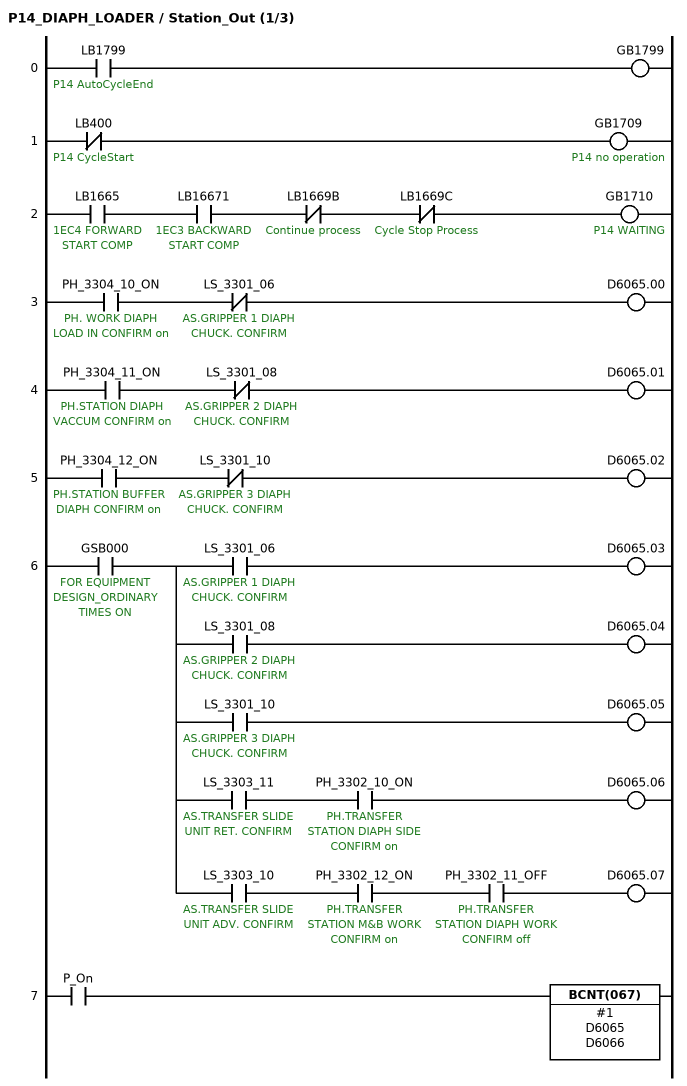
; [picture p216: P14_DIAPH_LOADER / Station_Out, rungs 0-7]
; rung 0
LD LB1799  ; P14 AutoCycleEnd
OUT GB1799
; rung 1
LDNOT LB400  ; P14 CycleStart
OUT GB1709  ; P14 no operation
; rung 2
LD LB1665  ; 1EC4 FORWARD START COMP
AND LB16671  ; 1EC3 BACKWARD START COMP
ANDNOT LB1669B  ; Continue process
ANDNOT LB1669C  ; Cycle Stop Process
OUT GB1710  ; P14 WAITING
; rung 3
LD PH_3304_10_ON  ; PH. WORK DIAPH LOAD IN CONFIRM on
ANDNOT LS_3301_06  ; AS.GRIPPER 1 DIAPH CHUCK. CONFIRM
OUT D6065.00
; rung 4
LD PH_3304_11_ON  ; PH.STATION DIAPH VACCUM CONFIRM on
ANDNOT LS_3301_08  ; AS.GRIPPER 2 DIAPH CHUCK. CONFIRM
OUT D6065.01
; rung 5
LD PH_3304_12_ON  ; PH.STATION BUFFER DIAPH CONFIRM on
ANDNOT LS_3301_10  ; AS.GRIPPER 3 DIAPH CHUCK. CONFIRM
OUT D6065.02
; rung 6
LD GSB000  ; FOR EQUIPMENT DESIGN_ORDINARY TIMES ON
OUT TR0
AND LS_3301_06  ; AS.GRIPPER 1 DIAPH CHUCK. CONFIRM
OUT D6065.03
LD TR0
AND LS_3301_08  ; AS.GRIPPER 2 DIAPH CHUCK. CONFIRM
OUT D6065.04
LD TR0
AND LS_3301_10  ; AS.GRIPPER 3 DIAPH CHUCK. CONFIRM
OUT D6065.05
LD TR0
AND LS_3303_11  ; AS.TRANSFER SLIDE UNIT RET. CONFIRM
AND PH_3302_10_ON  ; PH.TRANSFER STATION DIAPH SIDE CONFIRM on
OUT D6065.06
LD TR0
AND LS_3303_10  ; AS.TRANSFER SLIDE UNIT ADV. CONFIRM
AND PH_3302_12_ON  ; PH.TRANSFER STATION M&B WORK CONFIRM on
AND PH_3302_11_OFF  ; PH.TRANSFER STATION DIAPH WORK CONFIRM off
OUT D6065.07
; rung 7
LD P_On
BCNT(067) #1 D6065 D6066

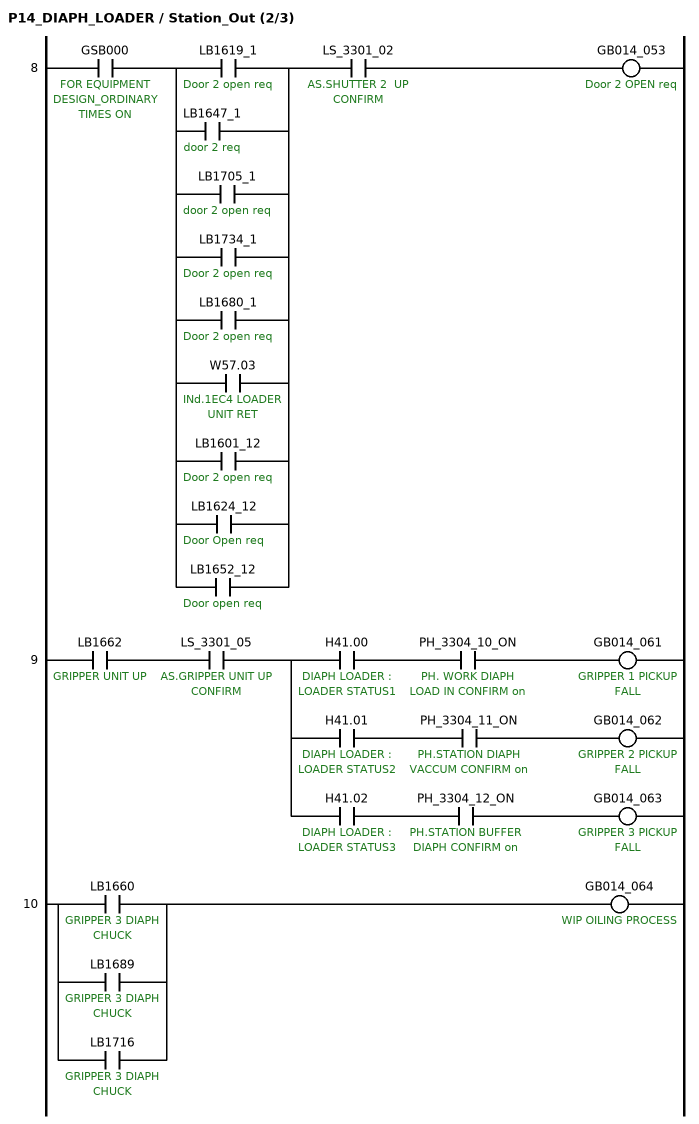
; rung 8
LD GSB000  ; FOR EQUIPMENT DESIGN_ORDINARY TIMES ON
LD LB1619_1  ; Door 2 open req
OR LB1647_1  ; door 2 req
OR LB1705_1  ; door 2 open req
OR LB1734_1  ; Door 2 open req
OR LB1680_1  ; Door 2 open req
OR W57.03  ; INd.1EC4 LOADER UNIT RET
OR LB1601_12  ; Door 2 open req
OR LB1624_12  ; Door Open req
OR LB1652_12  ; Door open req
ANDLD
AND LS_3301_02  ; AS.SHUTTER 2  UP CONFIRM
OUT GB014_053  ; Door 2 OPEN req
; rung 9
LD LB1662  ; GRIPPER UNIT UP
AND LS_3301_05  ; AS.GRIPPER UNIT UP CONFIRM
OUT TR0
AND H41.00  ; DIAPH LOADER : LOADER STATUS1
AND PH_3304_10_ON  ; PH. WORK DIAPH LOAD IN CONFIRM on
OUT GB014_061  ; GRIPPER 1 PICKUP FALL
LD TR0
AND H41.01  ; DIAPH LOADER : LOADER STATUS2
AND PH_3304_11_ON  ; PH.STATION DIAPH VACCUM CONFIRM on
OUT GB014_062  ; GRIPPER 2 PICKUP FALL
LD TR0
AND H41.02  ; DIAPH LOADER : LOADER STATUS3
AND PH_3304_12_ON  ; PH.STATION BUFFER DIAPH CONFIRM on
OUT GB014_063  ; GRIPPER 3 PICKUP FALL
; rung 10
LD LB1660  ; GRIPPER 3 DIAPH CHUCK
OR LB1689  ; GRIPPER 3 DIAPH CHUCK
OR LB1716  ; GRIPPER 3 DIAPH CHUCK
OUT GB014_064  ; WIP OILING PROCESS

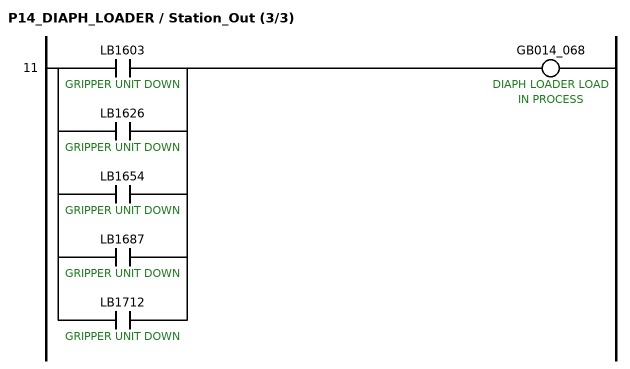
; rung 11
LD LB1603  ; GRIPPER UNIT DOWN
OR LB1626  ; GRIPPER UNIT DOWN
OR LB1654  ; GRIPPER UNIT DOWN
OR LB1687  ; GRIPPER UNIT DOWN
OR LB1712  ; GRIPPER UNIT DOWN
OUT GB014_068  ; DIAPH LOADER LOAD IN PROCESS

### Section Individual

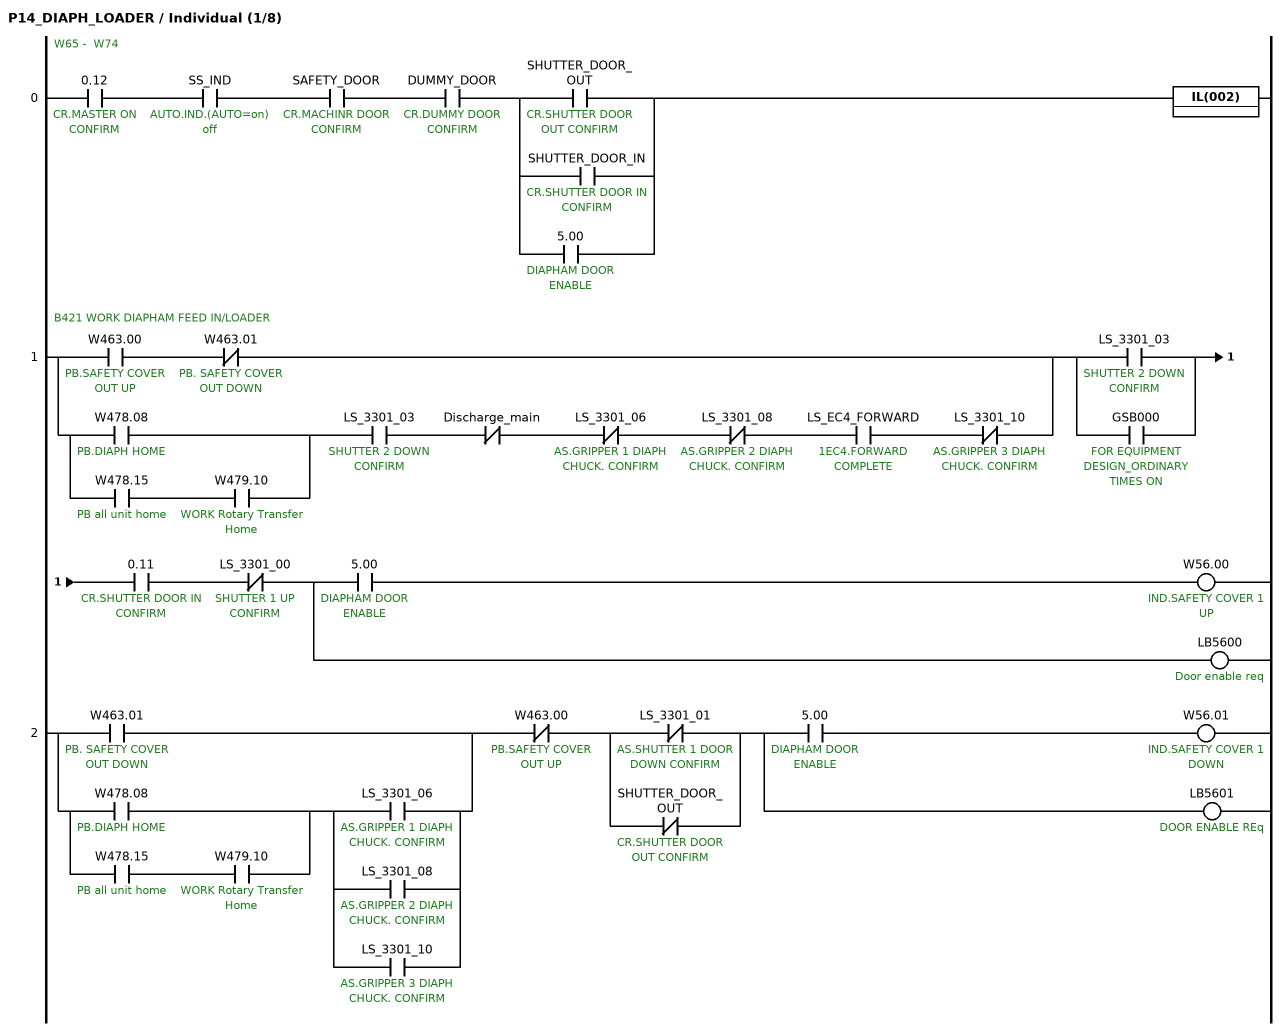
; rung 0: W65 -  W74
LD 0.12  ; CR.MASTER ON CONFIRM
AND SS_IND  ; AUTO.IND.(AUTO=on) off
AND SAFETY_DOOR  ; CR.MACHINR DOOR CONFIRM
AND DUMMY_DOOR  ; CR.DUMMY DOOR CONFIRM
LD SHUTTER_DOOR_OUT  ; CR.SHUTTER DOOR OUT CONFIRM
OR SHUTTER_DOOR_IN  ; CR.SHUTTER DOOR IN CONFIRM
OR 5.00  ; DIAPHAM DOOR ENABLE
ANDLD
IL(002)
; rung 1: B421 WORK DIAPHAM FEED IN/LOADER
LD W463.00  ; PB.SAFETY COVER OUT UP
ANDNOT W463.01  ; PB. SAFETY COVER OUT DOWN
LD W478.08  ; PB.DIAPH HOME
LD W478.15  ; PB all unit home
AND W479.10  ; WORK Rotary Transfer Home
ORLD
AND LS_3301_03  ; SHUTTER 2 DOWN CONFIRM
ANDNOT Discharge_main
ANDNOT LS_3301_06  ; AS.GRIPPER 1 DIAPH CHUCK. CONFIRM
ANDNOT LS_3301_08  ; AS.GRIPPER 2 DIAPH CHUCK. CONFIRM
AND LS_EC4_FORWARD  ; 1EC4.FORWARD COMPLETE
ANDNOT LS_3301_10  ; AS.GRIPPER 3 DIAPH CHUCK. CONFIRM
ORLD
LD LS_3301_03  ; SHUTTER 2 DOWN CONFIRM
OR GSB000  ; FOR EQUIPMENT DESIGN_ORDINARY TIMES ON
ANDLD
AND 0.11  ; CR.SHUTTER DOOR IN CONFIRM
ANDNOT LS_3301_00  ; SHUTTER 1 UP CONFIRM
OUT TR0
AND 5.00  ; DIAPHAM DOOR ENABLE
OUT W56.00  ; IND.SAFETY COVER 1 UP
LD TR0
OUT LB5600  ; Door enable req
; rung 2
LD W463.01  ; PB. SAFETY COVER OUT DOWN
LD W478.08  ; PB.DIAPH HOME
LD W478.15  ; PB all unit home
AND W479.10  ; WORK Rotary Transfer Home
ORLD
LD LS_3301_06  ; AS.GRIPPER 1 DIAPH CHUCK. CONFIRM
OR LS_3301_08  ; AS.GRIPPER 2 DIAPH CHUCK. CONFIRM
OR LS_3301_10  ; AS.GRIPPER 3 DIAPH CHUCK. CONFIRM
ANDLD
ORLD
ANDNOT W463.00  ; PB.SAFETY COVER OUT UP
LDNOT LS_3301_01  ; AS.SHUTTER 1 DOOR DOWN CONFIRM
ORNOT SHUTTER_DOOR_OUT  ; CR.SHUTTER DOOR OUT CONFIRM
ANDLD
OUT TR0
AND 5.00  ; DIAPHAM DOOR ENABLE
OUT W56.01  ; IND.SAFETY COVER 1 DOWN
LD TR0
OUT LB5601  ; DOOR ENABLE REq

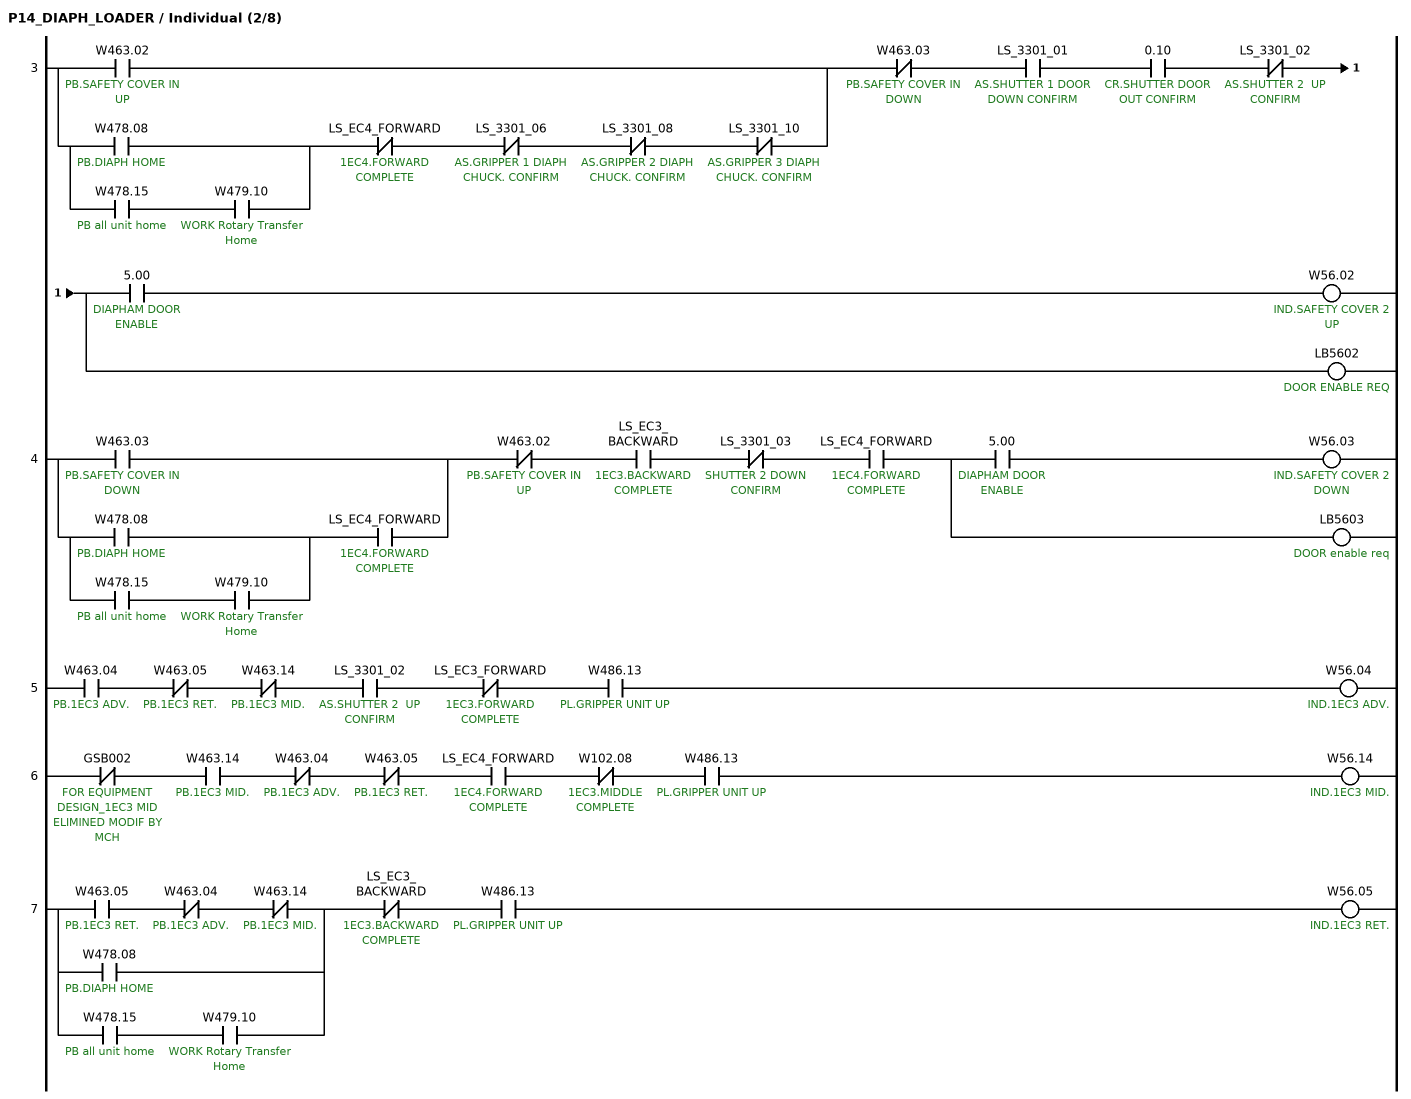
; rung 3
LD W463.02  ; PB.SAFETY COVER IN UP
LD W478.08  ; PB.DIAPH HOME
LD W478.15  ; PB all unit home
AND W479.10  ; WORK Rotary Transfer Home
ORLD
ANDNOT LS_EC4_FORWARD  ; 1EC4.FORWARD COMPLETE
ANDNOT LS_3301_06  ; AS.GRIPPER 1 DIAPH CHUCK. CONFIRM
ANDNOT LS_3301_08  ; AS.GRIPPER 2 DIAPH CHUCK. CONFIRM
ANDNOT LS_3301_10  ; AS.GRIPPER 3 DIAPH CHUCK. CONFIRM
ORLD
ANDNOT W463.03  ; PB.SAFETY COVER IN DOWN
AND LS_3301_01  ; AS.SHUTTER 1 DOOR DOWN CONFIRM
AND 0.10  ; CR.SHUTTER DOOR OUT CONFIRM
ANDNOT LS_3301_02  ; AS.SHUTTER 2  UP CONFIRM
OUT TR0
AND 5.00  ; DIAPHAM DOOR ENABLE
OUT W56.02  ; IND.SAFETY COVER 2 UP
LD TR0
OUT LB5602  ; DOOR ENABLE REQ
; rung 4
LD W463.03  ; PB.SAFETY COVER IN DOWN
LD W478.08  ; PB.DIAPH HOME
LD W478.15  ; PB all unit home
AND W479.10  ; WORK Rotary Transfer Home
ORLD
AND LS_EC4_FORWARD  ; 1EC4.FORWARD COMPLETE
ORLD
ANDNOT W463.02  ; PB.SAFETY COVER IN UP
AND LS_EC3_BACKWARD  ; 1EC3.BACKWARD COMPLETE
ANDNOT LS_3301_03  ; SHUTTER 2 DOWN CONFIRM
AND LS_EC4_FORWARD  ; 1EC4.FORWARD COMPLETE
OUT TR0
AND 5.00  ; DIAPHAM DOOR ENABLE
OUT W56.03  ; IND.SAFETY COVER 2 DOWN
LD TR0
OUT LB5603  ; DOOR enable req
; rung 5
LD W463.04  ; PB.1EC3 ADV.
ANDNOT W463.05  ; PB.1EC3 RET.
ANDNOT W463.14  ; PB.1EC3 MID.
AND LS_3301_02  ; AS.SHUTTER 2  UP CONFIRM
ANDNOT LS_EC3_FORWARD  ; 1EC3.FORWARD COMPLETE
AND W486.13  ; PL.GRIPPER UNIT UP
OUT W56.04  ; IND.1EC3 ADV.
; rung 6
LDNOT GSB002  ; FOR EQUIPMENT DESIGN_1EC3 MID ELIMINED MODIF BY MCH
AND W463.14  ; PB.1EC3 MID.
ANDNOT W463.04  ; PB.1EC3 ADV.
ANDNOT W463.05  ; PB.1EC3 RET.
AND LS_EC4_FORWARD  ; 1EC4.FORWARD COMPLETE
ANDNOT W102.08  ; 1EC3.MIDDLE COMPLETE
AND W486.13  ; PL.GRIPPER UNIT UP
OUT W56.14  ; IND.1EC3 MID.
; rung 7
LD W463.05  ; PB.1EC3 RET.
ANDNOT W463.04  ; PB.1EC3 ADV.
ANDNOT W463.14  ; PB.1EC3 MID.
LD W478.08  ; PB.DIAPH HOME
LD W478.15  ; PB all unit home
AND W479.10  ; WORK Rotary Transfer Home
ORLD
ORLD
ANDNOT LS_EC3_BACKWARD  ; 1EC3.BACKWARD COMPLETE
AND W486.13  ; PL.GRIPPER UNIT UP
OUT W56.05  ; IND.1EC3 RET.

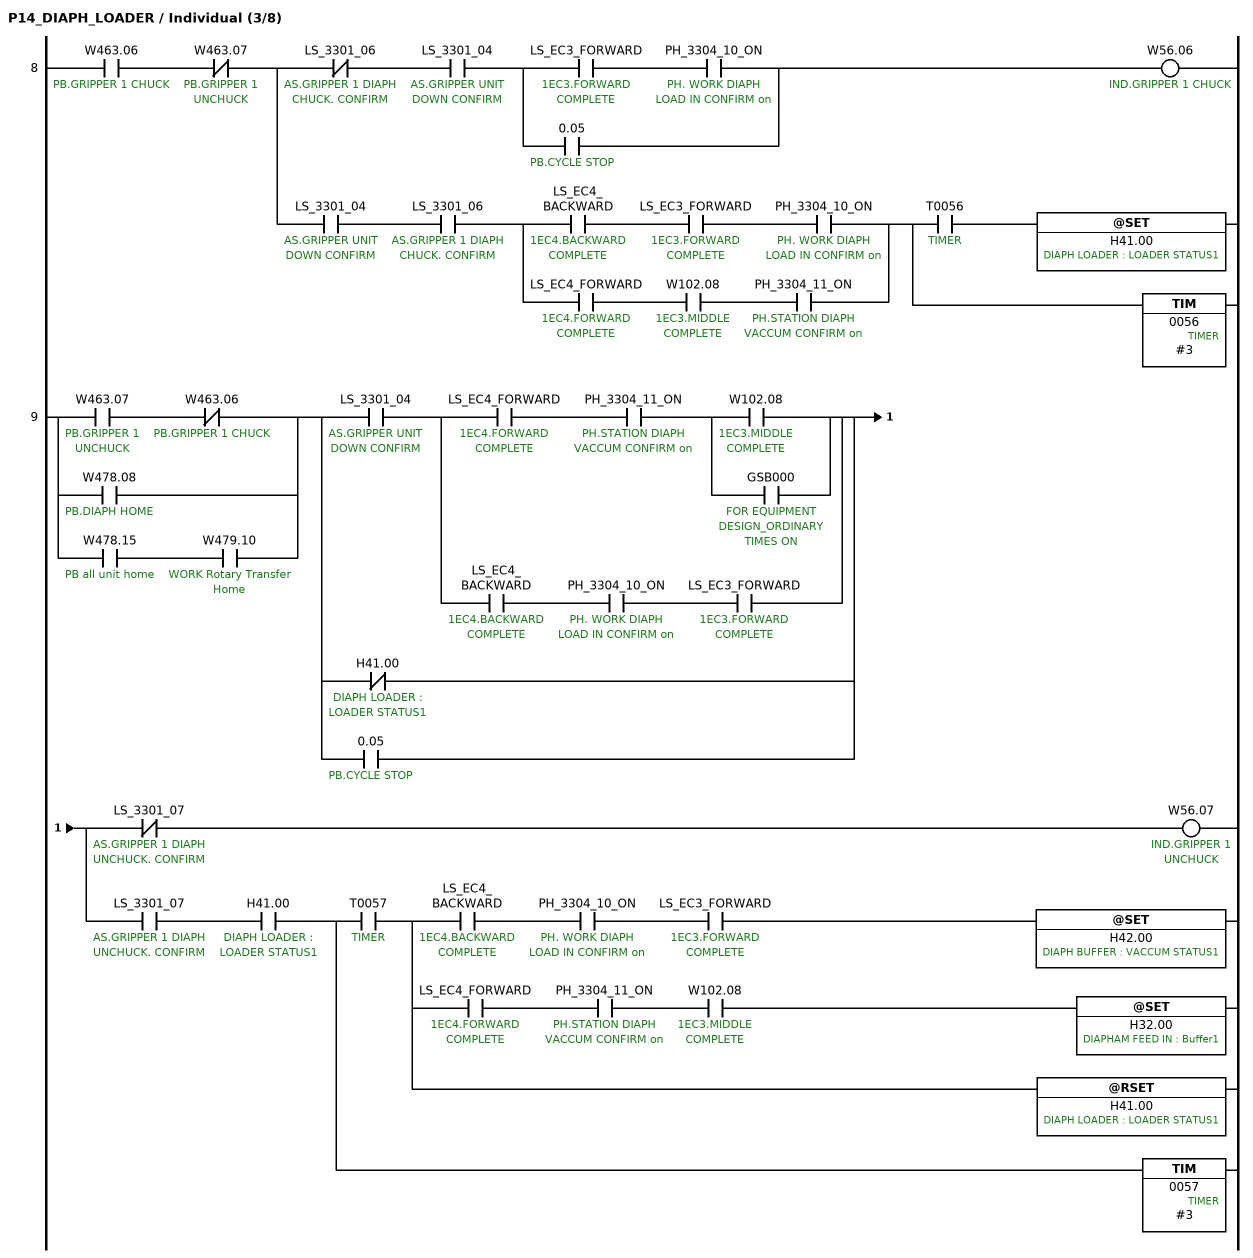
; rung 8
LD W463.06  ; PB.GRIPPER 1 CHUCK
ANDNOT W463.07  ; PB.GRIPPER 1 UNCHUCK
OUT TR0
ANDNOT LS_3301_06  ; AS.GRIPPER 1 DIAPH CHUCK. CONFIRM
AND LS_3301_04  ; AS.GRIPPER UNIT DOWN CONFIRM
LD LS_EC3_FORWARD  ; 1EC3.FORWARD COMPLETE
AND PH_3304_10_ON  ; PH. WORK DIAPH LOAD IN CONFIRM on
OR 0.05  ; PB.CYCLE STOP
ANDLD
OUT W56.06  ; IND.GRIPPER 1 CHUCK
LD TR0
AND LS_3301_04  ; AS.GRIPPER UNIT DOWN CONFIRM
AND LS_3301_06  ; AS.GRIPPER 1 DIAPH CHUCK. CONFIRM
LD LS_EC4_BACKWARD  ; 1EC4.BACKWARD COMPLETE
AND LS_EC3_FORWARD  ; 1EC3.FORWARD COMPLETE
AND PH_3304_10_ON  ; PH. WORK DIAPH LOAD IN CONFIRM on
LD LS_EC4_FORWARD  ; 1EC4.FORWARD COMPLETE
AND W102.08  ; 1EC3.MIDDLE COMPLETE
AND PH_3304_11_ON  ; PH.STATION DIAPH VACCUM CONFIRM on
ORLD
ANDLD
OUT TR0
AND T0056  ; TIMER
@SET H41.00  ; DIAPH LOADER : LOADER STATUS1
LD TR0
TIM 0056 #3  ; TIMER
; rung 9
LD W463.07  ; PB.GRIPPER 1 UNCHUCK
ANDNOT W463.06  ; PB.GRIPPER 1 CHUCK
OR W478.08  ; PB.DIAPH HOME
LD W478.15  ; PB all unit home
AND W479.10  ; WORK Rotary Transfer Home
ORLD
LD LS_3301_04  ; AS.GRIPPER UNIT DOWN CONFIRM
LD LS_EC4_FORWARD  ; 1EC4.FORWARD COMPLETE
AND PH_3304_11_ON  ; PH.STATION DIAPH VACCUM CONFIRM on
LD W102.08  ; 1EC3.MIDDLE COMPLETE
OR GSB000  ; FOR EQUIPMENT DESIGN_ORDINARY TIMES ON
ANDLD
LD LS_EC4_BACKWARD  ; 1EC4.BACKWARD COMPLETE
AND PH_3304_10_ON  ; PH. WORK DIAPH LOAD IN CONFIRM on
AND LS_EC3_FORWARD  ; 1EC3.FORWARD COMPLETE
ORLD
ANDLD
ORNOT H41.00  ; DIAPH LOADER : LOADER STATUS1
OR 0.05  ; PB.CYCLE STOP
ANDLD
OUT TR0
ANDNOT LS_3301_07  ; AS.GRIPPER 1 DIAPH UNCHUCK. CONFIRM
OUT W56.07  ; IND.GRIPPER 1 UNCHUCK
LD TR0
AND LS_3301_07  ; AS.GRIPPER 1 DIAPH UNCHUCK. CONFIRM
AND H41.00  ; DIAPH LOADER : LOADER STATUS1
OUT TR0
AND T0057  ; TIMER
OUT TR1
AND LS_EC4_BACKWARD  ; 1EC4.BACKWARD COMPLETE
AND PH_3304_10_ON  ; PH. WORK DIAPH LOAD IN CONFIRM on
AND LS_EC3_FORWARD  ; 1EC3.FORWARD COMPLETE
@SET H42.00  ; DIAPH BUFFER : VACCUM STATUS1
LD TR1
AND LS_EC4_FORWARD  ; 1EC4.FORWARD COMPLETE
AND PH_3304_11_ON  ; PH.STATION DIAPH VACCUM CONFIRM on
AND W102.08  ; 1EC3.MIDDLE COMPLETE
@SET H32.00  ; DIAPHAM FEED IN : Buffer1
LD TR1
@RSET H41.00  ; DIAPH LOADER : LOADER STATUS1
LD TR0
TIM 0057 #3  ; TIMER

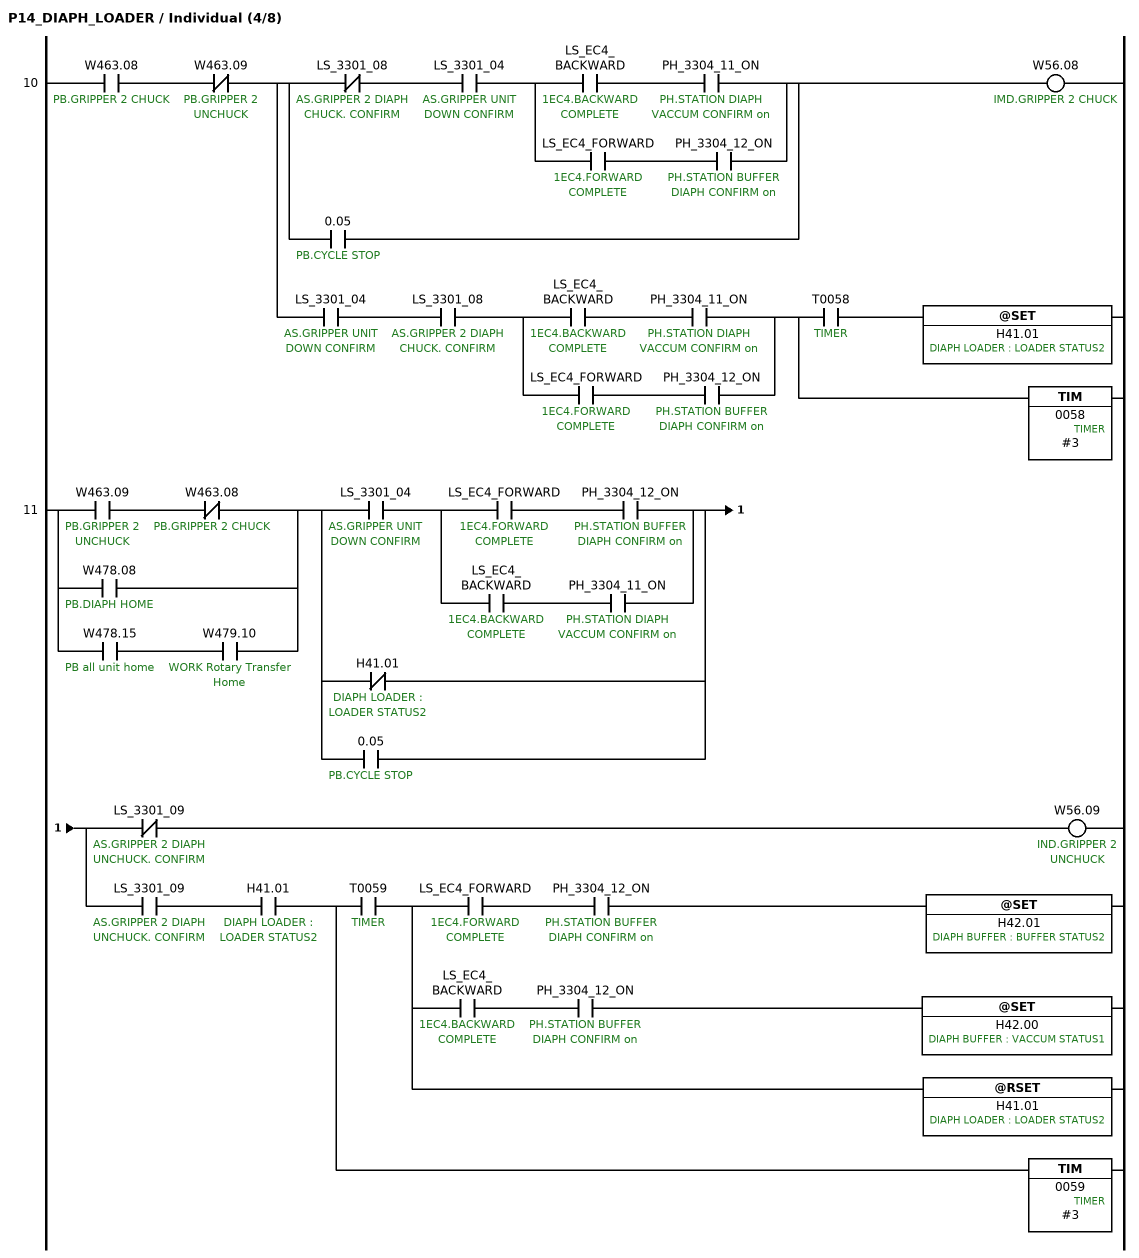
; rung 10
LD W463.08  ; PB.GRIPPER 2 CHUCK
ANDNOT W463.09  ; PB.GRIPPER 2 UNCHUCK
OUT TR0
LDNOT LS_3301_08  ; AS.GRIPPER 2 DIAPH CHUCK. CONFIRM
AND LS_3301_04  ; AS.GRIPPER UNIT DOWN CONFIRM
LD LS_EC4_BACKWARD  ; 1EC4.BACKWARD COMPLETE
AND PH_3304_11_ON  ; PH.STATION DIAPH VACCUM CONFIRM on
LD LS_EC4_FORWARD  ; 1EC4.FORWARD COMPLETE
AND PH_3304_12_ON  ; PH.STATION BUFFER DIAPH CONFIRM on
ORLD
ANDLD
OR 0.05  ; PB.CYCLE STOP
ANDLD
OUT W56.08  ; IMD.GRIPPER 2 CHUCK
LD TR0
AND LS_3301_04  ; AS.GRIPPER UNIT DOWN CONFIRM
AND LS_3301_08  ; AS.GRIPPER 2 DIAPH CHUCK. CONFIRM
LD LS_EC4_BACKWARD  ; 1EC4.BACKWARD COMPLETE
AND PH_3304_11_ON  ; PH.STATION DIAPH VACCUM CONFIRM on
LD LS_EC4_FORWARD  ; 1EC4.FORWARD COMPLETE
AND PH_3304_12_ON  ; PH.STATION BUFFER DIAPH CONFIRM on
ORLD
ANDLD
OUT TR0
AND T0058  ; TIMER
@SET H41.01  ; DIAPH LOADER : LOADER STATUS2
LD TR0
TIM 0058 #3  ; TIMER
; rung 11
LD W463.09  ; PB.GRIPPER 2 UNCHUCK
ANDNOT W463.08  ; PB.GRIPPER 2 CHUCK
OR W478.08  ; PB.DIAPH HOME
LD W478.15  ; PB all unit home
AND W479.10  ; WORK Rotary Transfer Home
ORLD
LD LS_3301_04  ; AS.GRIPPER UNIT DOWN CONFIRM
LD LS_EC4_FORWARD  ; 1EC4.FORWARD COMPLETE
AND PH_3304_12_ON  ; PH.STATION BUFFER DIAPH CONFIRM on
LD LS_EC4_BACKWARD  ; 1EC4.BACKWARD COMPLETE
AND PH_3304_11_ON  ; PH.STATION DIAPH VACCUM CONFIRM on
ORLD
ANDLD
ORNOT H41.01  ; DIAPH LOADER : LOADER STATUS2
OR 0.05  ; PB.CYCLE STOP
ANDLD
OUT TR0
ANDNOT LS_3301_09  ; AS.GRIPPER 2 DIAPH UNCHUCK. CONFIRM
OUT W56.09  ; IND.GRIPPER 2 UNCHUCK
LD TR0
AND LS_3301_09  ; AS.GRIPPER 2 DIAPH UNCHUCK. CONFIRM
AND H41.01  ; DIAPH LOADER : LOADER STATUS2
OUT TR0
AND T0059  ; TIMER
OUT TR1
AND LS_EC4_FORWARD  ; 1EC4.FORWARD COMPLETE
AND PH_3304_12_ON  ; PH.STATION BUFFER DIAPH CONFIRM on
@SET H42.01  ; DIAPH BUFFER : BUFFER STATUS2
LD TR1
AND LS_EC4_BACKWARD  ; 1EC4.BACKWARD COMPLETE
AND PH_3304_12_ON  ; PH.STATION BUFFER DIAPH CONFIRM on
@SET H42.00  ; DIAPH BUFFER : VACCUM STATUS1
LD TR1
@RSET H41.01  ; DIAPH LOADER : LOADER STATUS2
LD TR0
TIM 0059 #3  ; TIMER

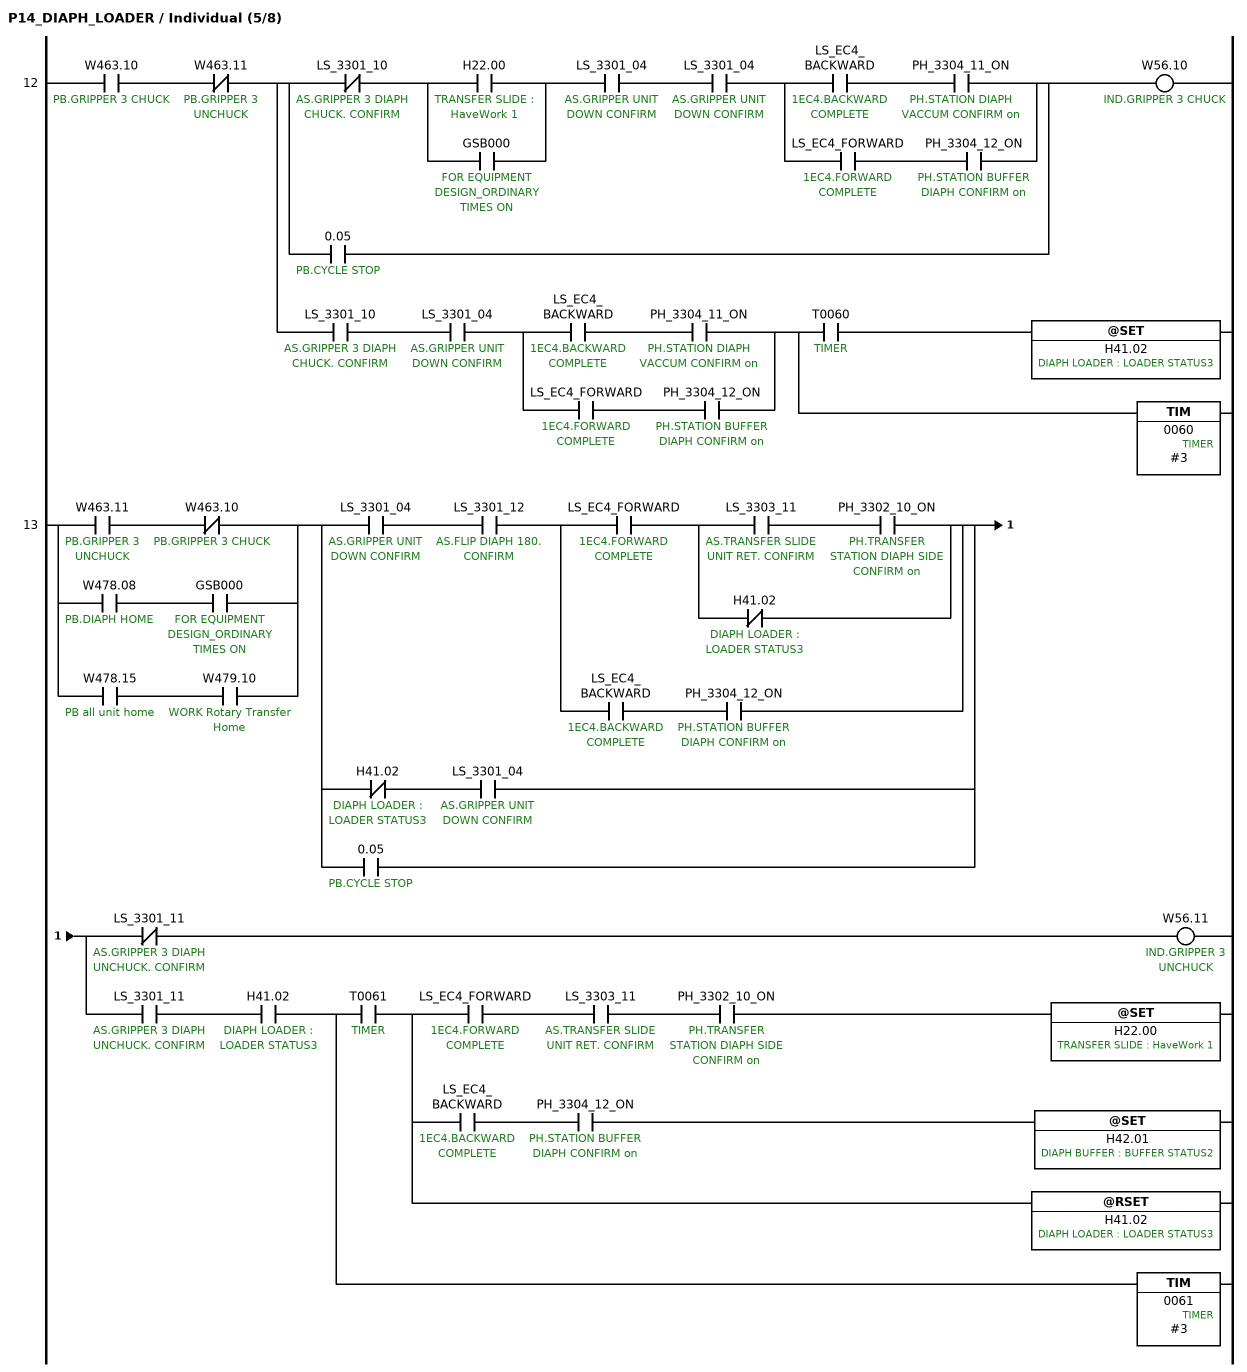
; rung 12
LD W463.10  ; PB.GRIPPER 3 CHUCK
ANDNOT W463.11  ; PB.GRIPPER 3 UNCHUCK
OUT TR0
LDNOT LS_3301_10  ; AS.GRIPPER 3 DIAPH CHUCK. CONFIRM
LD H22.00  ; TRANSFER SLIDE : HaveWork 1
OR GSB000  ; FOR EQUIPMENT DESIGN_ORDINARY TIMES ON
ANDLD
AND LS_3301_04  ; AS.GRIPPER UNIT DOWN CONFIRM  // PROHIBIT LOAD WORK FORM TRANSFER UNIT
AND LS_3301_04  ; AS.GRIPPER UNIT DOWN CONFIRM
LD LS_EC4_BACKWARD  ; 1EC4.BACKWARD COMPLETE
AND PH_3304_11_ON  ; PH.STATION DIAPH VACCUM CONFIRM on
LD LS_EC4_FORWARD  ; 1EC4.FORWARD COMPLETE
AND PH_3304_12_ON  ; PH.STATION BUFFER DIAPH CONFIRM on
ORLD
ANDLD
OR 0.05  ; PB.CYCLE STOP
ANDLD
OUT W56.10  ; IND.GRIPPER 3 CHUCK
LD TR0
AND LS_3301_10  ; AS.GRIPPER 3 DIAPH CHUCK. CONFIRM
AND LS_3301_04  ; AS.GRIPPER UNIT DOWN CONFIRM
LD LS_EC4_BACKWARD  ; 1EC4.BACKWARD COMPLETE
AND PH_3304_11_ON  ; PH.STATION DIAPH VACCUM CONFIRM on
LD LS_EC4_FORWARD  ; 1EC4.FORWARD COMPLETE
AND PH_3304_12_ON  ; PH.STATION BUFFER DIAPH CONFIRM on
ORLD
ANDLD
OUT TR0
AND T0060  ; TIMER
@SET H41.02  ; DIAPH LOADER : LOADER STATUS3
LD TR0
TIM 0060 #3  ; TIMER
; rung 13
LD W463.11  ; PB.GRIPPER 3 UNCHUCK
ANDNOT W463.10  ; PB.GRIPPER 3 CHUCK
LD W478.08  ; PB.DIAPH HOME
AND GSB000  ; FOR EQUIPMENT DESIGN_ORDINARY TIMES ON
ORLD
LD W478.15  ; PB all unit home
AND W479.10  ; WORK Rotary Transfer Home
ORLD
LD LS_3301_04  ; AS.GRIPPER UNIT DOWN CONFIRM
AND LS_3301_12  ; AS.FLIP DIAPH 180. CONFIRM
LD LS_EC4_FORWARD  ; 1EC4.FORWARD COMPLETE
LD LS_3303_11  ; AS.TRANSFER SLIDE UNIT RET. CONFIRM
AND PH_3302_10_ON  ; PH.TRANSFER STATION DIAPH SIDE CONFIRM on
ORNOT H41.02  ; DIAPH LOADER : LOADER STATUS3
ANDLD
LD LS_EC4_BACKWARD  ; 1EC4.BACKWARD COMPLETE
AND PH_3304_12_ON  ; PH.STATION BUFFER DIAPH CONFIRM on
ORLD
ANDLD
LDNOT H41.02  ; DIAPH LOADER : LOADER STATUS3
AND LS_3301_04  ; AS.GRIPPER UNIT DOWN CONFIRM
ORLD
OR 0.05  ; PB.CYCLE STOP
ANDLD
OUT TR0
ANDNOT LS_3301_11  ; AS.GRIPPER 3 DIAPH UNCHUCK. CONFIRM
OUT W56.11  ; IND.GRIPPER 3 UNCHUCK
LD TR0
AND LS_3301_11  ; AS.GRIPPER 3 DIAPH UNCHUCK. CONFIRM
AND H41.02  ; DIAPH LOADER : LOADER STATUS3
OUT TR0
AND T0061  ; TIMER
OUT TR1
AND LS_EC4_FORWARD  ; 1EC4.FORWARD COMPLETE
AND LS_3303_11  ; AS.TRANSFER SLIDE UNIT RET. CONFIRM
AND PH_3302_10_ON  ; PH.TRANSFER STATION DIAPH SIDE CONFIRM on
@SET H22.00  ; TRANSFER SLIDE : HaveWork 1
LD TR1
AND LS_EC4_BACKWARD  ; 1EC4.BACKWARD COMPLETE
AND PH_3304_12_ON  ; PH.STATION BUFFER DIAPH CONFIRM on
@SET H42.01  ; DIAPH BUFFER : BUFFER STATUS2
LD TR1
@RSET H41.02  ; DIAPH LOADER : LOADER STATUS3
LD TR0
TIM 0061 #3  ; TIMER

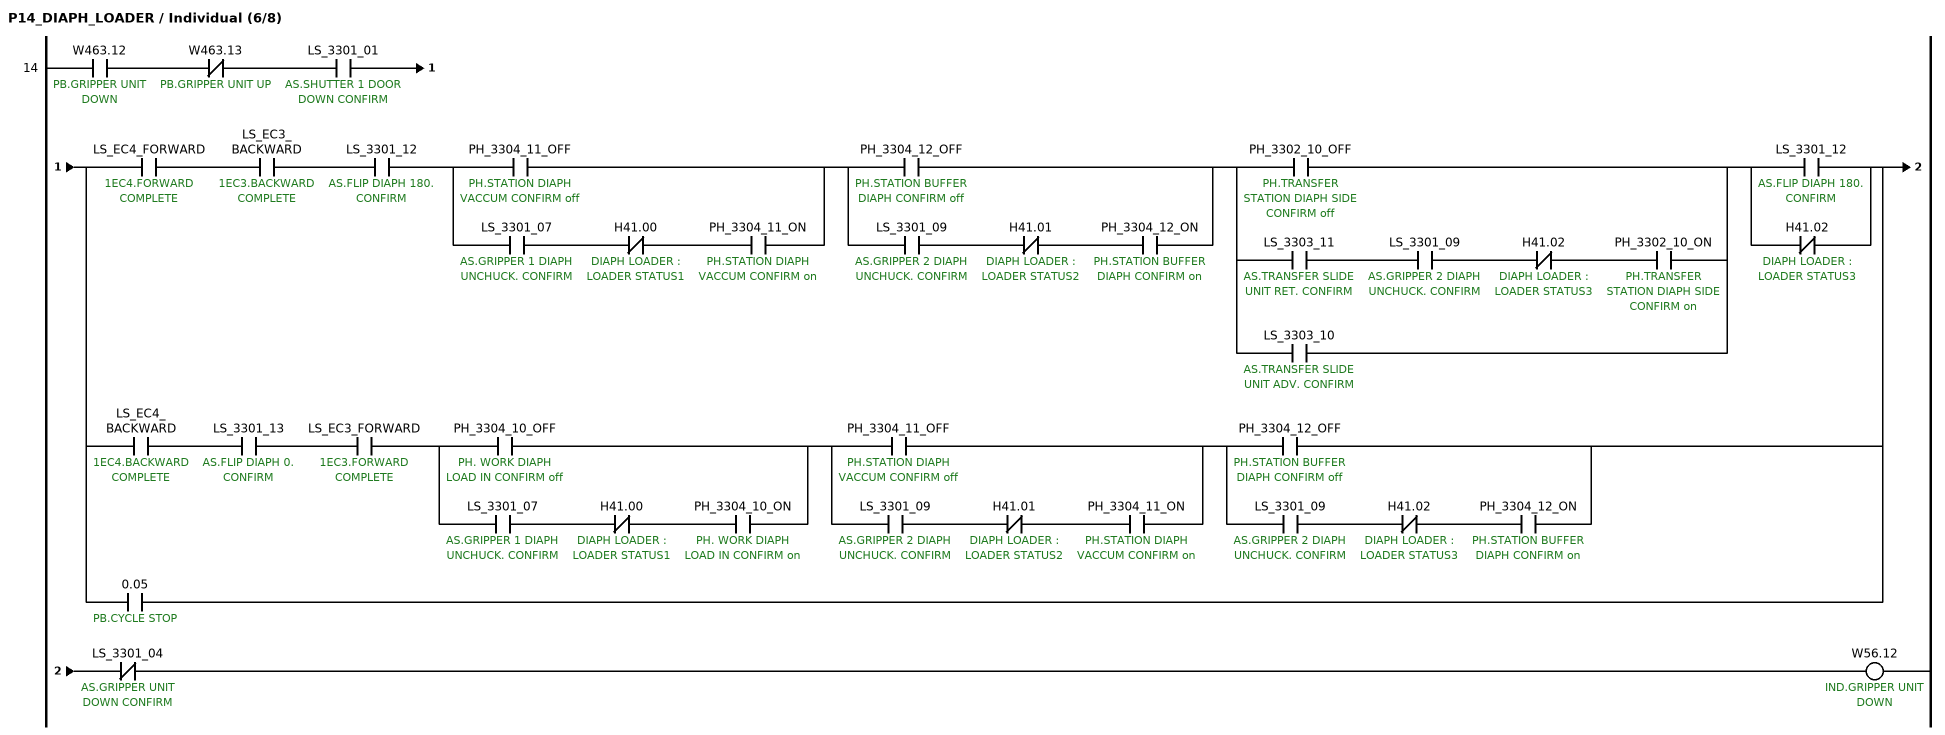
; rung 14
LD W463.12  ; PB.GRIPPER UNIT DOWN
ANDNOT W463.13  ; PB.GRIPPER UNIT UP
AND LS_3301_01  ; AS.SHUTTER 1 DOOR DOWN CONFIRM
LD LS_EC4_FORWARD  ; 1EC4.FORWARD COMPLETE
AND LS_EC3_BACKWARD  ; 1EC3.BACKWARD COMPLETE
AND LS_3301_12  ; AS.FLIP DIAPH 180. CONFIRM
LD PH_3304_11_OFF  ; PH.STATION DIAPH VACCUM CONFIRM off
LD LS_3301_07  ; AS.GRIPPER 1 DIAPH UNCHUCK. CONFIRM
ANDNOT H41.00  ; DIAPH LOADER : LOADER STATUS1
AND PH_3304_11_ON  ; PH.STATION DIAPH VACCUM CONFIRM on
ORLD
ANDLD
LD PH_3304_12_OFF  ; PH.STATION BUFFER DIAPH CONFIRM off
LD LS_3301_09  ; AS.GRIPPER 2 DIAPH UNCHUCK. CONFIRM
ANDNOT H41.01  ; DIAPH LOADER : LOADER STATUS2
AND PH_3304_12_ON  ; PH.STATION BUFFER DIAPH CONFIRM on
ORLD
ANDLD
LD PH_3302_10_OFF  ; PH.TRANSFER STATION DIAPH SIDE CONFIRM off
LD LS_3303_11  ; AS.TRANSFER SLIDE UNIT RET. CONFIRM
AND LS_3301_09  ; AS.GRIPPER 2 DIAPH UNCHUCK. CONFIRM
ANDNOT H41.02  ; DIAPH LOADER : LOADER STATUS3
AND PH_3302_10_ON  ; PH.TRANSFER STATION DIAPH SIDE CONFIRM on
ORLD
OR LS_3303_10  ; AS.TRANSFER SLIDE UNIT ADV. CONFIRM
ANDLD
LD LS_3301_12  ; AS.FLIP DIAPH 180. CONFIRM
ORNOT H41.02  ; DIAPH LOADER : LOADER STATUS3
ANDLD
LD LS_EC4_BACKWARD  ; 1EC4.BACKWARD COMPLETE
AND LS_3301_13  ; AS.FLIP DIAPH 0. CONFIRM
AND LS_EC3_FORWARD  ; 1EC3.FORWARD COMPLETE
LD PH_3304_10_OFF  ; PH. WORK DIAPH LOAD IN CONFIRM off
LD LS_3301_07  ; AS.GRIPPER 1 DIAPH UNCHUCK. CONFIRM
ANDNOT H41.00  ; DIAPH LOADER : LOADER STATUS1
AND PH_3304_10_ON  ; PH. WORK DIAPH LOAD IN CONFIRM on
ORLD
ANDLD
LD PH_3304_11_OFF  ; PH.STATION DIAPH VACCUM CONFIRM off
LD LS_3301_09  ; AS.GRIPPER 2 DIAPH UNCHUCK. CONFIRM
ANDNOT H41.01  ; DIAPH LOADER : LOADER STATUS2
AND PH_3304_11_ON  ; PH.STATION DIAPH VACCUM CONFIRM on
ORLD
ANDLD
LD PH_3304_12_OFF  ; PH.STATION BUFFER DIAPH CONFIRM off
LD LS_3301_09  ; AS.GRIPPER 2 DIAPH UNCHUCK. CONFIRM
ANDNOT H41.02  ; DIAPH LOADER : LOADER STATUS3
AND PH_3304_12_ON  ; PH.STATION BUFFER DIAPH CONFIRM on
ORLD
ANDLD
ORLD
OR 0.05  ; PB.CYCLE STOP
ANDLD
ANDNOT LS_3301_04  ; AS.GRIPPER UNIT DOWN CONFIRM
OUT W56.12  ; IND.GRIPPER UNIT DOWN

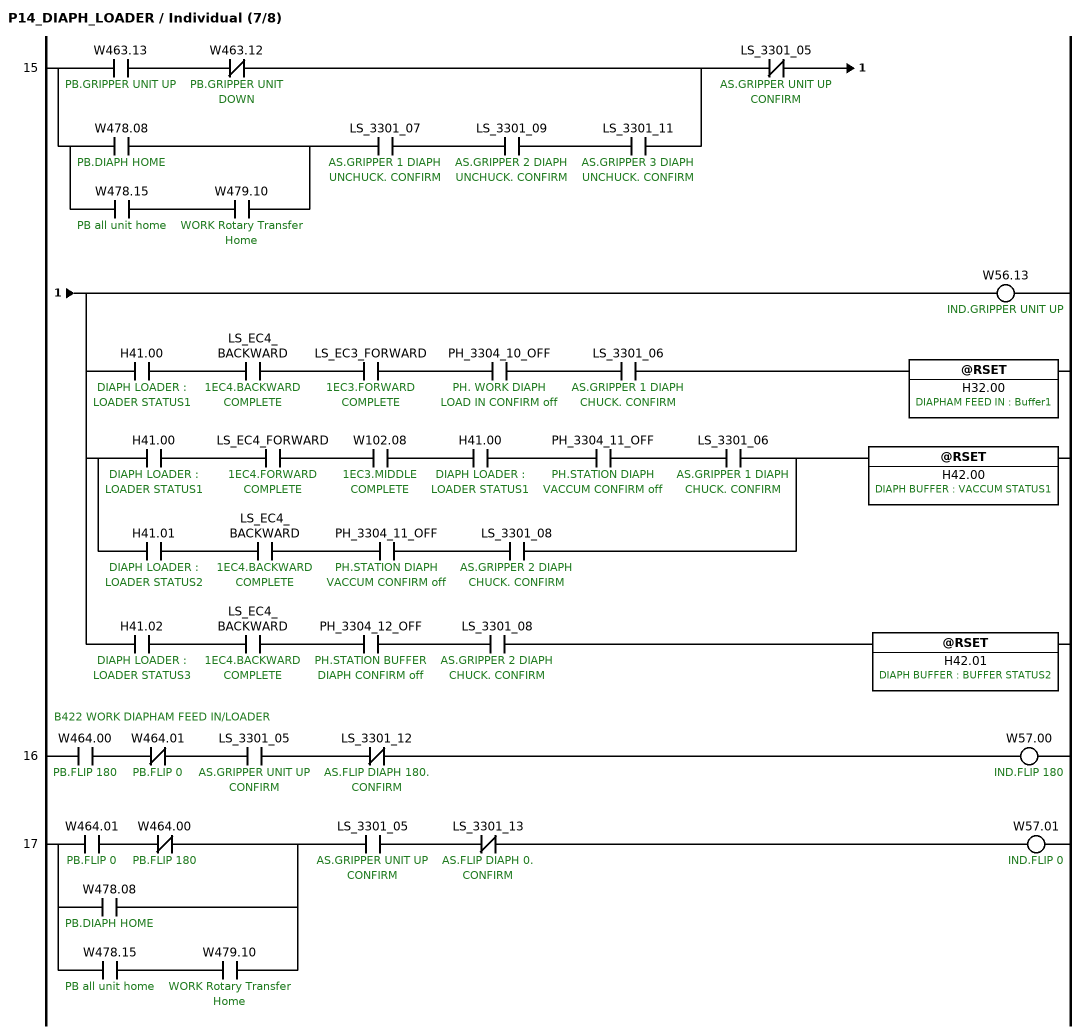
; rung 15
LD W463.13  ; PB.GRIPPER UNIT UP
ANDNOT W463.12  ; PB.GRIPPER UNIT DOWN
LD W478.08  ; PB.DIAPH HOME
LD W478.15  ; PB all unit home
AND W479.10  ; WORK Rotary Transfer Home
ORLD
AND LS_3301_07  ; AS.GRIPPER 1 DIAPH UNCHUCK. CONFIRM
AND LS_3301_09  ; AS.GRIPPER 2 DIAPH UNCHUCK. CONFIRM
AND LS_3301_11  ; AS.GRIPPER 3 DIAPH UNCHUCK. CONFIRM
ORLD
ANDNOT LS_3301_05  ; AS.GRIPPER UNIT UP CONFIRM
OUT TR0
OUT W56.13  ; IND.GRIPPER UNIT UP
AND H41.00  ; DIAPH LOADER : LOADER STATUS1
AND LS_EC4_BACKWARD  ; 1EC4.BACKWARD COMPLETE
AND LS_EC3_FORWARD  ; 1EC3.FORWARD COMPLETE
AND PH_3304_10_OFF  ; PH. WORK DIAPH LOAD IN CONFIRM off
AND LS_3301_06  ; AS.GRIPPER 1 DIAPH CHUCK. CONFIRM
@RSET H32.00  ; DIAPHAM FEED IN : Buffer1
LD TR0
LD H41.00  ; DIAPH LOADER : LOADER STATUS1
AND LS_EC4_FORWARD  ; 1EC4.FORWARD COMPLETE
AND W102.08  ; 1EC3.MIDDLE COMPLETE
AND H41.00  ; DIAPH LOADER : LOADER STATUS1
AND PH_3304_11_OFF  ; PH.STATION DIAPH VACCUM CONFIRM off
AND LS_3301_06  ; AS.GRIPPER 1 DIAPH CHUCK. CONFIRM
LD H41.01  ; DIAPH LOADER : LOADER STATUS2
AND LS_EC4_BACKWARD  ; 1EC4.BACKWARD COMPLETE
AND PH_3304_11_OFF  ; PH.STATION DIAPH VACCUM CONFIRM off
AND LS_3301_08  ; AS.GRIPPER 2 DIAPH CHUCK. CONFIRM
ORLD
ANDLD
@RSET H42.00  ; DIAPH BUFFER : VACCUM STATUS1
LD TR0
AND H41.02  ; DIAPH LOADER : LOADER STATUS3
AND LS_EC4_BACKWARD  ; 1EC4.BACKWARD COMPLETE
AND PH_3304_12_OFF  ; PH.STATION BUFFER DIAPH CONFIRM off
AND LS_3301_08  ; AS.GRIPPER 2 DIAPH CHUCK. CONFIRM
@RSET H42.01  ; DIAPH BUFFER : BUFFER STATUS2
; rung 16: B422 WORK DIAPHAM FEED IN/LOADER
LD W464.00  ; PB.FLIP 180
ANDNOT W464.01  ; PB.FLIP 0
AND LS_3301_05  ; AS.GRIPPER UNIT UP CONFIRM
ANDNOT LS_3301_12  ; AS.FLIP DIAPH 180. CONFIRM
OUT W57.00  ; IND.FLIP 180
; rung 17
LD W464.01  ; PB.FLIP 0
ANDNOT W464.00  ; PB.FLIP 180
OR W478.08  ; PB.DIAPH HOME
LD W478.15  ; PB all unit home
AND W479.10  ; WORK Rotary Transfer Home
ORLD
AND LS_3301_05  ; AS.GRIPPER UNIT UP CONFIRM
ANDNOT LS_3301_13  ; AS.FLIP DIAPH 0. CONFIRM
OUT W57.01  ; IND.FLIP 0

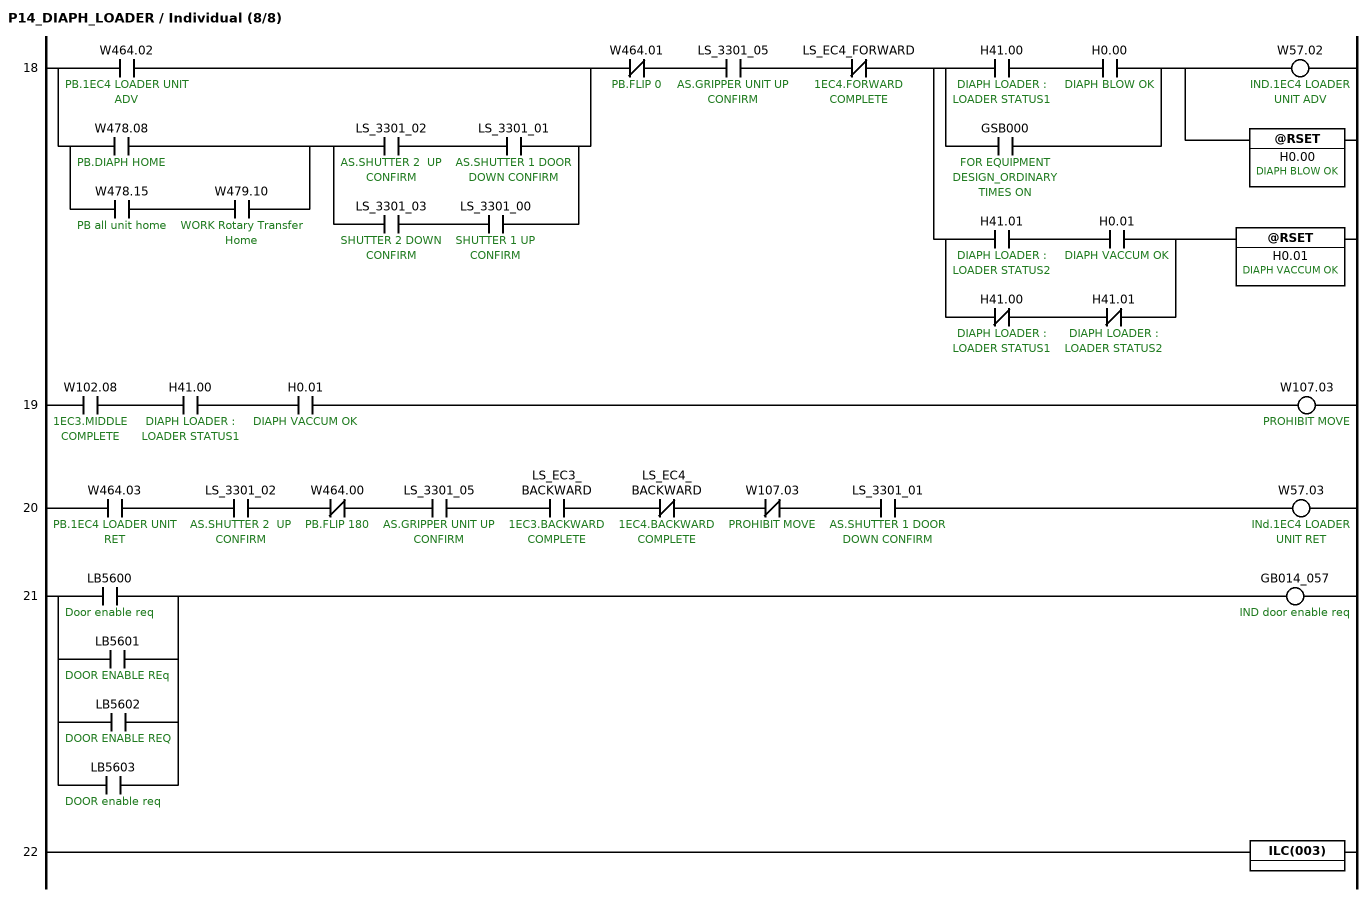
; rung 18
LD W464.02  ; PB.1EC4 LOADER UNIT ADV
LD W478.08  ; PB.DIAPH HOME
LD W478.15  ; PB all unit home
AND W479.10  ; WORK Rotary Transfer Home
ORLD
LD LS_3301_02  ; AS.SHUTTER 2  UP CONFIRM
AND LS_3301_01  ; AS.SHUTTER 1 DOOR DOWN CONFIRM
LD LS_3301_03  ; SHUTTER 2 DOWN CONFIRM
AND LS_3301_00  ; SHUTTER 1 UP CONFIRM
ORLD
ANDLD
ORLD
ANDNOT W464.01  ; PB.FLIP 0
AND LS_3301_05  ; AS.GRIPPER UNIT UP CONFIRM
ANDNOT LS_EC4_FORWARD  ; 1EC4.FORWARD COMPLETE
OUT TR0
LD H41.00  ; DIAPH LOADER : LOADER STATUS1
AND H0.00  ; DIAPH BLOW OK
OR GSB000  ; FOR EQUIPMENT DESIGN_ORDINARY TIMES ON
ANDLD
OUT W57.02  ; IND.1EC4 LOADER UNIT ADV
@RSET H0.00  ; DIAPH BLOW OK
LD TR0
LD H41.01  ; DIAPH LOADER : LOADER STATUS2
AND H0.01  ; DIAPH VACCUM OK
LDNOT H41.00  ; DIAPH LOADER : LOADER STATUS1
ANDNOT H41.01  ; DIAPH LOADER : LOADER STATUS2
ORLD
ANDLD
@RSET H0.01  ; DIAPH VACCUM OK
; rung 19
LD W102.08  ; 1EC3.MIDDLE COMPLETE
AND H41.00  ; DIAPH LOADER : LOADER STATUS1
AND H0.01  ; DIAPH VACCUM OK
OUT W107.03  ; PROHIBIT MOVE
; rung 20
LD W464.03  ; PB.1EC4 LOADER UNIT RET
AND LS_3301_02  ; AS.SHUTTER 2  UP CONFIRM
ANDNOT W464.00  ; PB.FLIP 180
AND LS_3301_05  ; AS.GRIPPER UNIT UP CONFIRM
AND LS_EC3_BACKWARD  ; 1EC3.BACKWARD COMPLETE
ANDNOT LS_EC4_BACKWARD  ; 1EC4.BACKWARD COMPLETE
ANDNOT W107.03  ; PROHIBIT MOVE
AND LS_3301_01  ; AS.SHUTTER 1 DOOR DOWN CONFIRM
OUT W57.03  ; INd.1EC4 LOADER UNIT RET
; rung 21
LD LB5600  ; Door enable req
OR LB5601  ; DOOR ENABLE REq
OR LB5602  ; DOOR ENABLE REQ
OR LB5603  ; DOOR enable req
OUT GB014_057  ; IND door enable req
; rung 22
ILC(003)

### Section END
; rung 0
END(001)

## Program P15_SLIDE_TRANSFER (cyclic task 5)
Local symbols
LB1799 E0_26.14 BOOL  ; P14 AutoCycleEnd
LB1800 E0_26.15 BOOL  ; AUTO START BEGIN
LB1801 E0_30.00 BOOL  ; MemoryInterlockCondition
LB1802 E0_30.01 BOOL  ; TRANSFER SLIDE UNIT ADV
LB1803 E0_30.02 BOOL  ; TRANSFER SLIDE UNIT ADV CONF
LB1804 E0_30.03 BOOL  ; TRANSFER SLIDE UNIT RET
LB1805 E0_30.04 BOOL  ; TRANSFER SLIDE UNIT RET CONF
LB1900 E0_30.05 BOOL  ; 1cycle start
LB1999 E0_30.06 BOOL  ; P15 AutoCycleEnd
LB340 E0_30.07 BOOL  ; IND 1 CYCLE
LB500 E0_30.08 BOOL  ; P15 CycleStart
LB501 E0_30.09 BOOL  ; P15 SLIDE ADV.
LB502 E0_30.10 BOOL  ; P15 Slide return

### Section HMI_Output

### Section Autorun

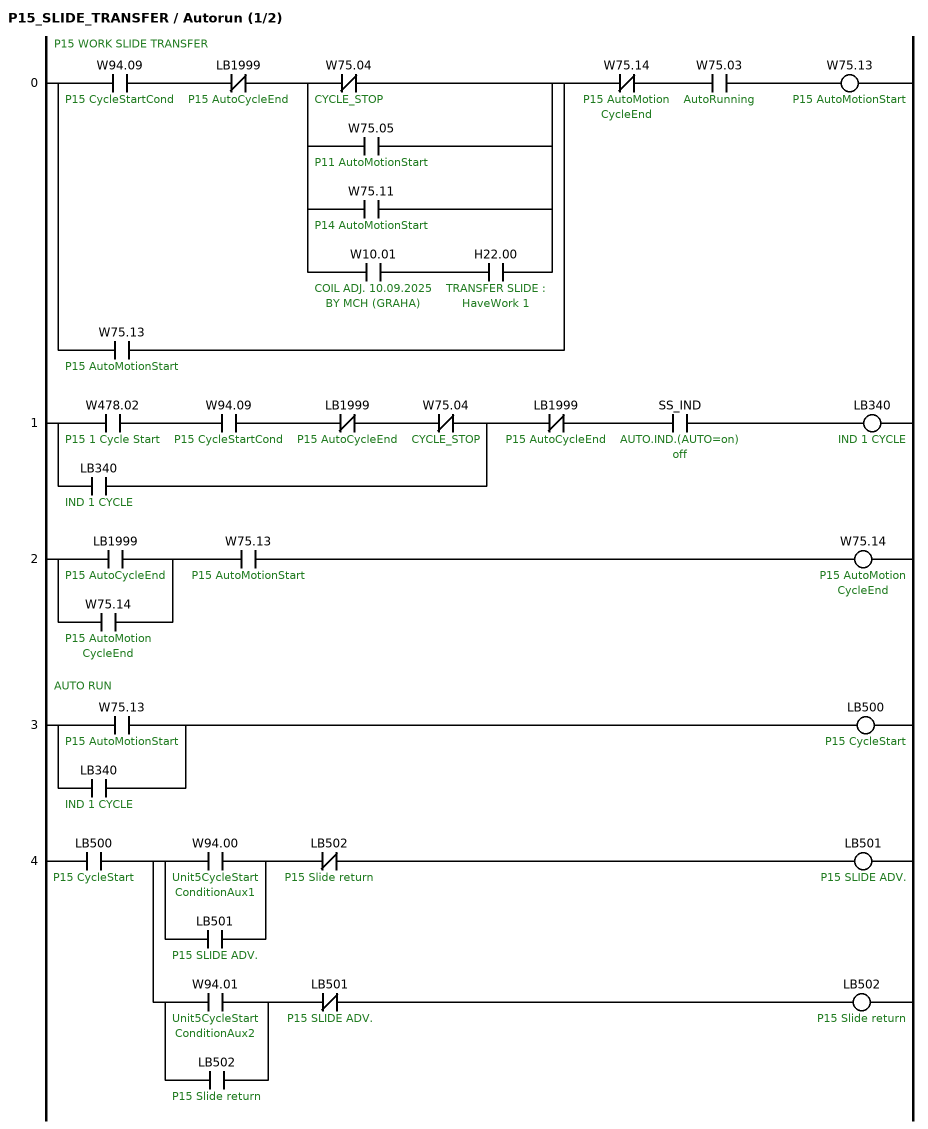
; rung 0: P15 WORK SLIDE TRANSFER
LD W94.09  ; P15 CycleStartCond
ANDNOT LB1999  ; P15 AutoCycleEnd
LDNOT W75.04  ; CYCLE_STOP
OR W75.05  ; P11 AutoMotionStart
OR W75.11  ; P14 AutoMotionStart
LD W10.01  ; COIL ADJ. 10.09.2025 BY MCH (GRAHA)
AND H22.00  ; TRANSFER SLIDE : HaveWork 1
ORLD
ANDLD
OR W75.13  ; P15 AutoMotionStart
ANDNOT W75.14  ; P15 AutoMotion CycleEnd
AND W75.03  ; AutoRunning
OUT W75.13  ; P15 AutoMotionStart
; rung 1
LD W478.02  ; P15 1 Cycle Start
AND W94.09  ; P15 CycleStartCond
ANDNOT LB1999  ; P15 AutoCycleEnd
ANDNOT W75.04  ; CYCLE_STOP
OR LB340  ; IND 1 CYCLE
ANDNOT LB1999  ; P15 AutoCycleEnd
AND SS_IND  ; AUTO.IND.(AUTO=on) off
OUT LB340  ; IND 1 CYCLE
; rung 2
LD LB1999  ; P15 AutoCycleEnd
OR W75.14  ; P15 AutoMotion CycleEnd
AND W75.13  ; P15 AutoMotionStart
OUT W75.14  ; P15 AutoMotion CycleEnd
; rung 3: AUTO RUN
LD W75.13  ; P15 AutoMotionStart
OR LB340  ; IND 1 CYCLE
OUT LB500  ; P15 CycleStart
; rung 4
LD LB500  ; P15 CycleStart
OUT TR0
LD W94.00  ; Unit5CycleStartConditionAux1
OR LB501  ; P15 SLIDE ADV.
ANDLD
ANDNOT LB502  ; P15 Slide return
OUT LB501  ; P15 SLIDE ADV.
LD TR0
LD W94.01  ; Unit5CycleStartConditionAux2
OR LB502  ; P15 Slide return
ANDLD
ANDNOT LB501  ; P15 SLIDE ADV.
OUT LB502  ; P15 Slide return

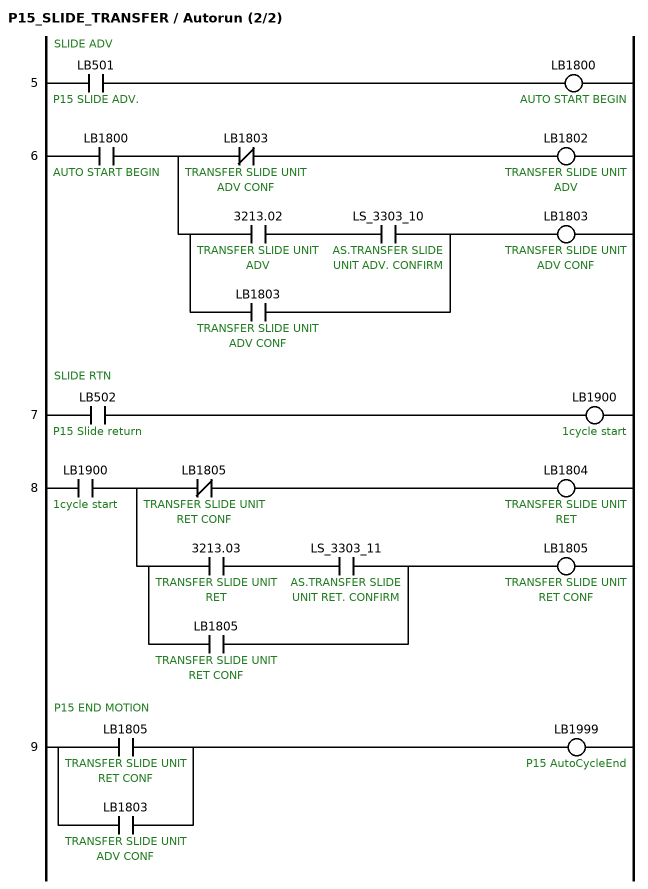
; rung 5: SLIDE ADV
LD LB501  ; P15 SLIDE ADV.
OUT LB1800  ; AUTO START BEGIN
; rung 6
LD LB1800  ; AUTO START BEGIN
OUT TR0
ANDNOT LB1803  ; TRANSFER SLIDE UNIT ADV CONF
OUT LB1802  ; TRANSFER SLIDE UNIT ADV
LD TR0
LD 3213.02  ; TRANSFER SLIDE UNIT ADV
AND LS_3303_10  ; AS.TRANSFER SLIDE UNIT ADV. CONFIRM
OR LB1803  ; TRANSFER SLIDE UNIT ADV CONF
ANDLD
OUT LB1803  ; TRANSFER SLIDE UNIT ADV CONF
; rung 7: SLIDE RTN
LD LB502  ; P15 Slide return
OUT LB1900  ; 1cycle start
; rung 8
LD LB1900  ; 1cycle start
OUT TR0
ANDNOT LB1805  ; TRANSFER SLIDE UNIT RET CONF
OUT LB1804  ; TRANSFER SLIDE UNIT RET
LD TR0
LD 3213.03  ; TRANSFER SLIDE UNIT RET
AND LS_3303_11  ; AS.TRANSFER SLIDE UNIT RET. CONFIRM
OR LB1805  ; TRANSFER SLIDE UNIT RET CONF
ANDLD
OUT LB1805  ; TRANSFER SLIDE UNIT RET CONF
; rung 9: P15 END MOTION
LD LB1805  ; TRANSFER SLIDE UNIT RET CONF
OR LB1803  ; TRANSFER SLIDE UNIT ADV CONF
OUT LB1999  ; P15 AutoCycleEnd

### Section Condition

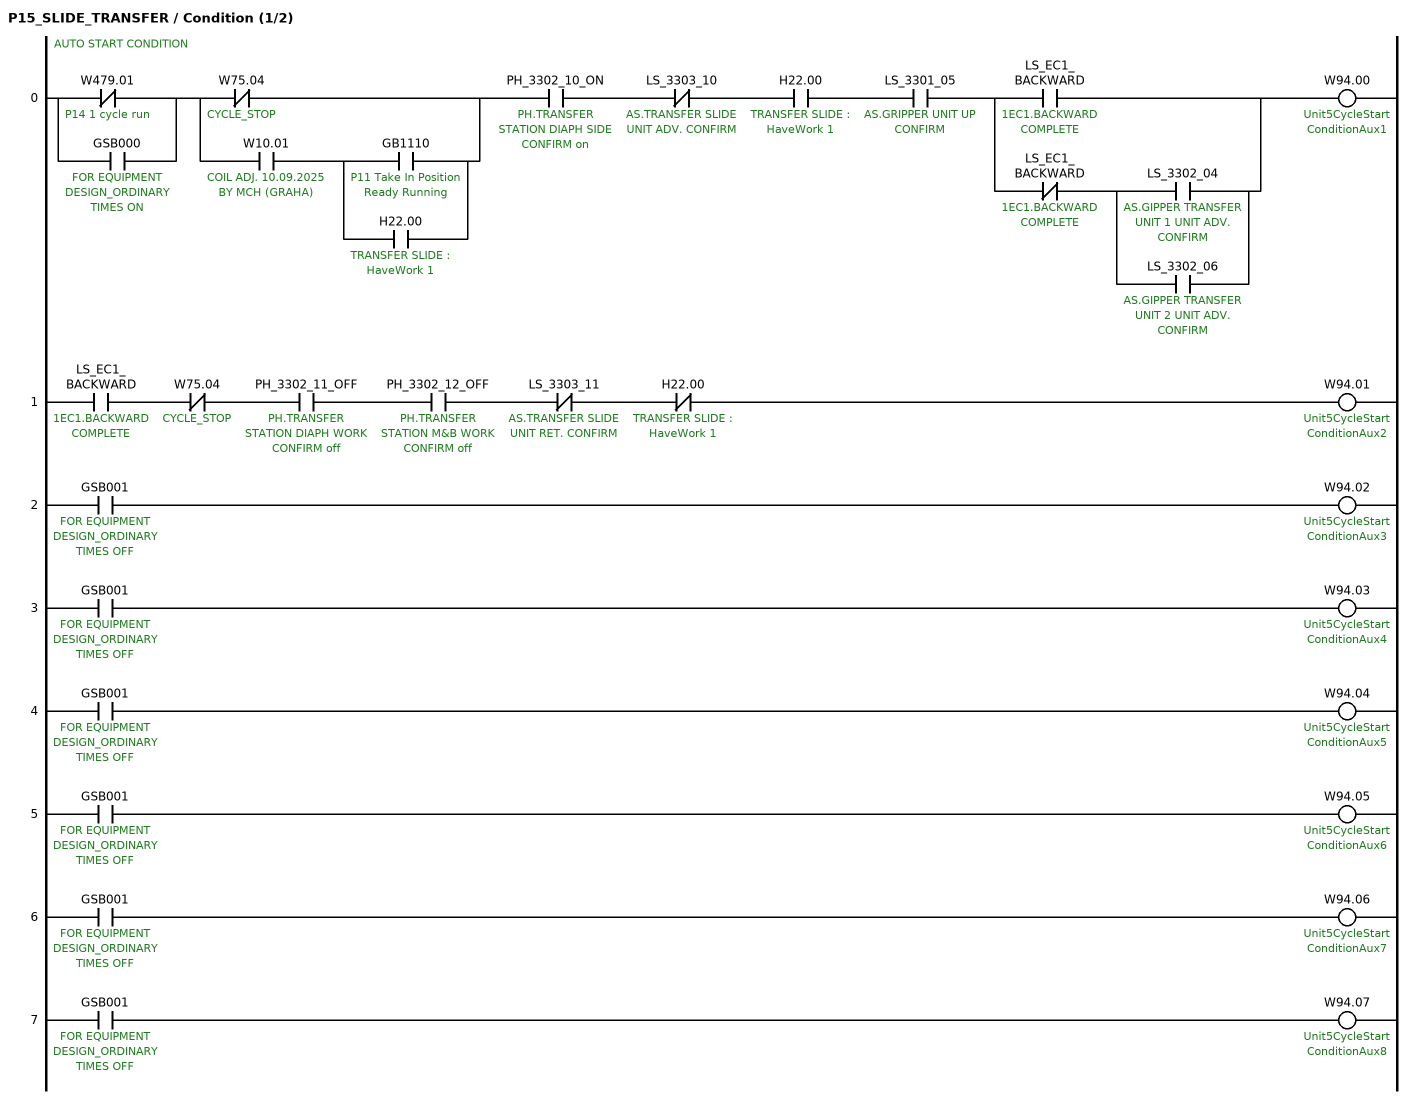
; rung 0: AUTO START CONDITION
LDNOT W479.01  ; P14 1 cycle run
OR GSB000  ; FOR EQUIPMENT DESIGN_ORDINARY TIMES ON
LDNOT W75.04  ; CYCLE_STOP
LD W10.01  ; COIL ADJ. 10.09.2025 BY MCH (GRAHA)
LD GB1110  ; P11 Take In Position Ready Running
OR H22.00  ; TRANSFER SLIDE : HaveWork 1
ANDLD
ORLD
ANDLD
AND PH_3302_10_ON  ; PH.TRANSFER STATION DIAPH SIDE CONFIRM on
ANDNOT LS_3303_10  ; AS.TRANSFER SLIDE UNIT ADV. CONFIRM
AND H22.00  ; TRANSFER SLIDE : HaveWork 1
AND LS_3301_05  ; AS.GRIPPER UNIT UP CONFIRM
LD LS_EC1_BACKWARD  ; 1EC1.BACKWARD COMPLETE
LDNOT LS_EC1_BACKWARD  ; 1EC1.BACKWARD COMPLETE
LD LS_3302_04  ; AS.GIPPER TRANSFER UNIT 1 UNIT ADV. CONFIRM
OR LS_3302_06  ; AS.GIPPER TRANSFER UNIT 2 UNIT ADV. CONFIRM
ANDLD
ORLD
ANDLD
OUT W94.00  ; Unit5CycleStartConditionAux1
; rung 1
LD LS_EC1_BACKWARD  ; 1EC1.BACKWARD COMPLETE
ANDNOT W75.04  ; CYCLE_STOP
AND PH_3302_11_OFF  ; PH.TRANSFER STATION DIAPH WORK CONFIRM off
AND PH_3302_12_OFF  ; PH.TRANSFER STATION M&B WORK CONFIRM off
ANDNOT LS_3303_11  ; AS.TRANSFER SLIDE UNIT RET. CONFIRM
ANDNOT H22.00  ; TRANSFER SLIDE : HaveWork 1
OUT W94.01  ; Unit5CycleStartConditionAux2
; rung 2
LD GSB001  ; FOR EQUIPMENT DESIGN_ORDINARY TIMES OFF
OUT W94.02  ; Unit5CycleStartConditionAux3
; rung 3
LD GSB001  ; FOR EQUIPMENT DESIGN_ORDINARY TIMES OFF
OUT W94.03  ; Unit5CycleStartConditionAux4
; rung 4
LD GSB001  ; FOR EQUIPMENT DESIGN_ORDINARY TIMES OFF
OUT W94.04  ; Unit5CycleStartConditionAux5
; rung 5
LD GSB001  ; FOR EQUIPMENT DESIGN_ORDINARY TIMES OFF
OUT W94.05  ; Unit5CycleStartConditionAux6
; rung 6
LD GSB001  ; FOR EQUIPMENT DESIGN_ORDINARY TIMES OFF
OUT W94.06  ; Unit5CycleStartConditionAux7
; rung 7
LD GSB001  ; FOR EQUIPMENT DESIGN_ORDINARY TIMES OFF
OUT W94.07  ; Unit5CycleStartConditionAux8

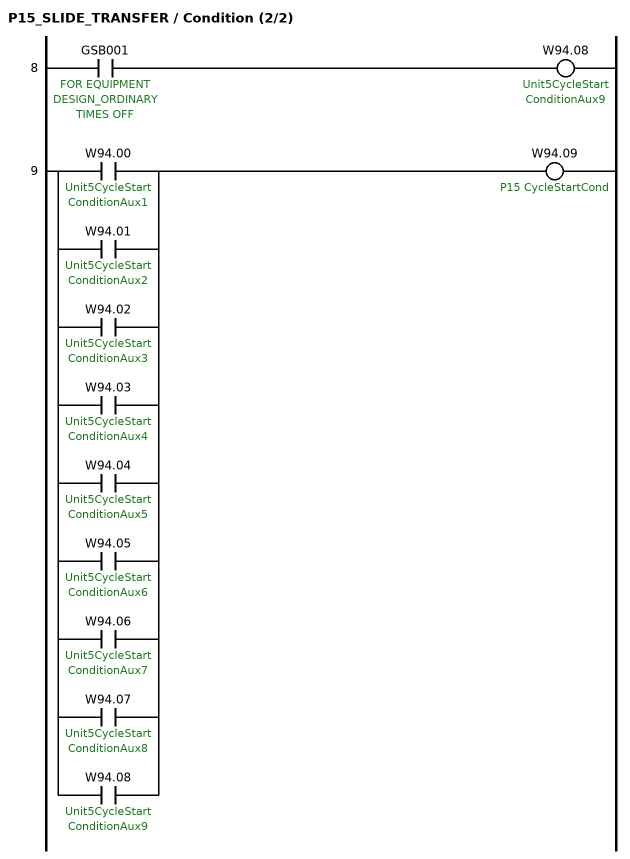
; rung 8
LD GSB001  ; FOR EQUIPMENT DESIGN_ORDINARY TIMES OFF
OUT W94.08  ; Unit5CycleStartConditionAux9
; rung 9
LD W94.00  ; Unit5CycleStartConditionAux1
OR W94.01  ; Unit5CycleStartConditionAux2
OR W94.02  ; Unit5CycleStartConditionAux3
OR W94.03  ; Unit5CycleStartConditionAux4
OR W94.04  ; Unit5CycleStartConditionAux5
OR W94.05  ; Unit5CycleStartConditionAux6
OR W94.06  ; Unit5CycleStartConditionAux7
OR W94.07  ; Unit5CycleStartConditionAux8
OR W94.08  ; Unit5CycleStartConditionAux9
OUT W94.09  ; P15 CycleStartCond

### Section Device_Output

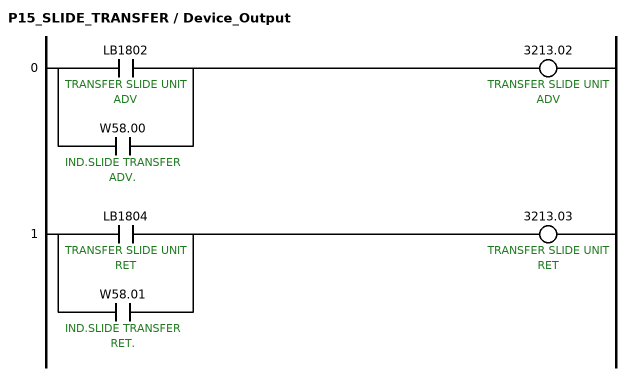
; rung 0
LD LB1802  ; TRANSFER SLIDE UNIT ADV
OR W58.00  ; IND.SLIDE TRANSFER ADV.
OUT 3213.02  ; TRANSFER SLIDE UNIT ADV
; rung 1
LD LB1804  ; TRANSFER SLIDE UNIT RET
OR W58.01  ; IND.SLIDE TRANSFER RET.
OUT 3213.03  ; TRANSFER SLIDE UNIT RET

### Section Station_Output

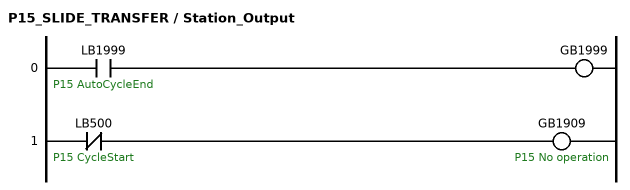
; rung 0
LD LB1999  ; P15 AutoCycleEnd
OUT GB1999
; rung 1
LDNOT LB500  ; P15 CycleStart
OUT GB1909  ; P15 No operation

### Section Individual

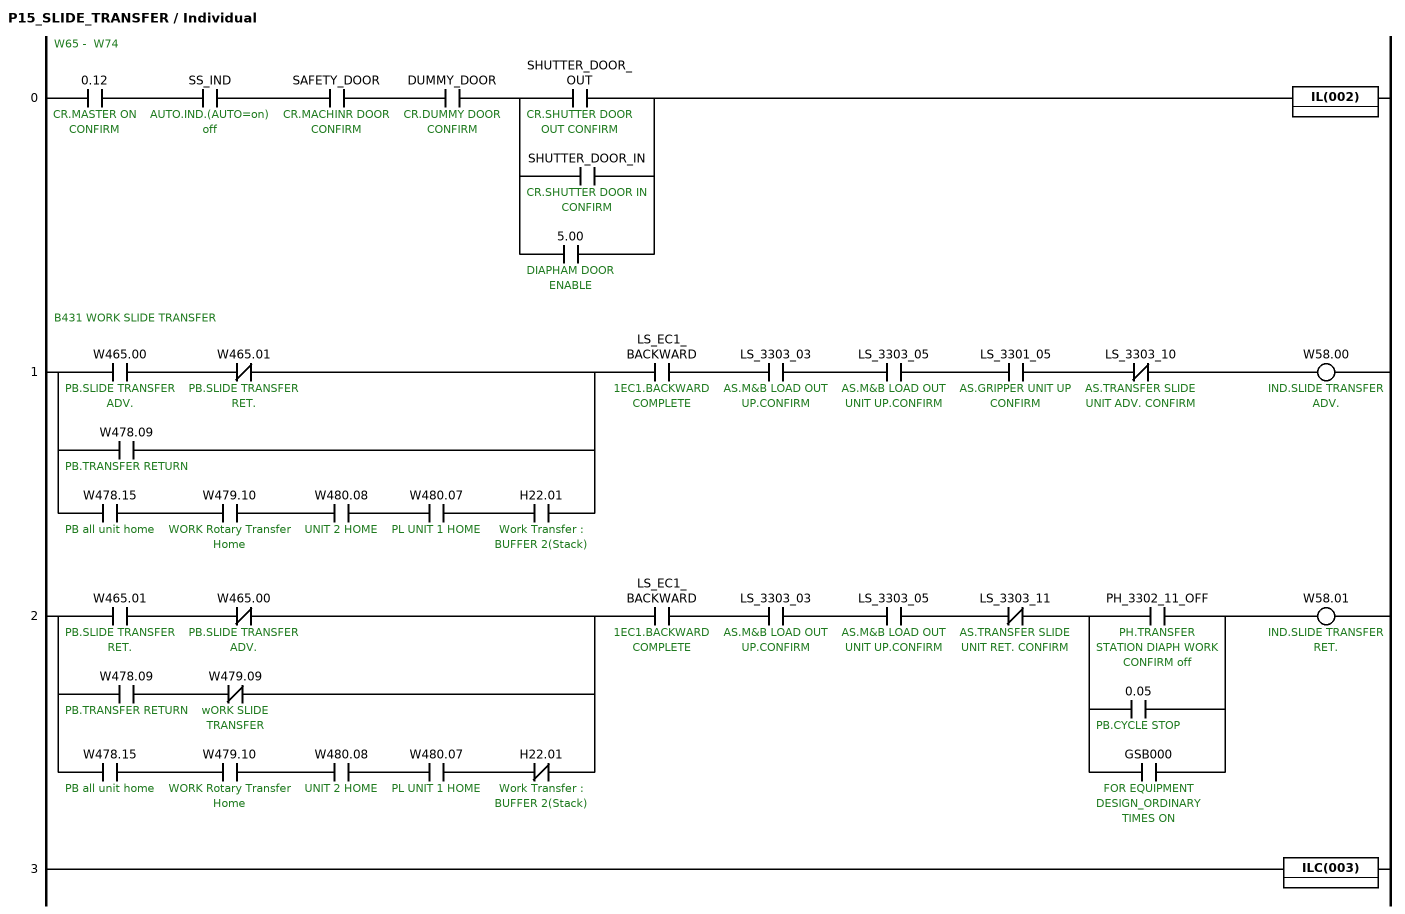
; rung 0: W65 -  W74
LD 0.12  ; CR.MASTER ON CONFIRM
AND SS_IND  ; AUTO.IND.(AUTO=on) off
AND SAFETY_DOOR  ; CR.MACHINR DOOR CONFIRM
AND DUMMY_DOOR  ; CR.DUMMY DOOR CONFIRM
LD SHUTTER_DOOR_OUT  ; CR.SHUTTER DOOR OUT CONFIRM
OR SHUTTER_DOOR_IN  ; CR.SHUTTER DOOR IN CONFIRM
OR 5.00  ; DIAPHAM DOOR ENABLE
ANDLD
IL(002)
; rung 1: B431 WORK SLIDE TRANSFER
LD W465.00  ; PB.SLIDE TRANSFER ADV.
ANDNOT W465.01  ; PB.SLIDE TRANSFER RET.
OR W478.09  ; PB.TRANSFER RETURN
LD W478.15  ; PB all unit home
AND W479.10  ; WORK Rotary Transfer Home
AND W480.08  ; UNIT 2 HOME
AND W480.07  ; PL UNIT 1 HOME
AND H22.01  ; Work Transfer : BUFFER 2(Stack)
ORLD
AND LS_EC1_BACKWARD  ; 1EC1.BACKWARD COMPLETE
AND LS_3303_03  ; AS.M&B LOAD OUT UP.CONFIRM
AND LS_3303_05  ; AS.M&B LOAD OUT UNIT UP.CONFIRM
AND LS_3301_05  ; AS.GRIPPER UNIT UP CONFIRM
ANDNOT LS_3303_10  ; AS.TRANSFER SLIDE UNIT ADV. CONFIRM
OUT W58.00  ; IND.SLIDE TRANSFER ADV.
; rung 2
LD W465.01  ; PB.SLIDE TRANSFER RET.
ANDNOT W465.00  ; PB.SLIDE TRANSFER ADV.
LD W478.09  ; PB.TRANSFER RETURN
ANDNOT W479.09  ; wORK SLIDE TRANSFER
ORLD
LD W478.15  ; PB all unit home
AND W479.10  ; WORK Rotary Transfer Home
AND W480.08  ; UNIT 2 HOME
AND W480.07  ; PL UNIT 1 HOME
ANDNOT H22.01  ; Work Transfer : BUFFER 2(Stack)
ORLD
AND LS_EC1_BACKWARD  ; 1EC1.BACKWARD COMPLETE
AND LS_3303_03  ; AS.M&B LOAD OUT UP.CONFIRM
AND LS_3303_05  ; AS.M&B LOAD OUT UNIT UP.CONFIRM
ANDNOT LS_3303_11  ; AS.TRANSFER SLIDE UNIT RET. CONFIRM
LD PH_3302_11_OFF  ; PH.TRANSFER STATION DIAPH WORK CONFIRM off
OR 0.05  ; PB.CYCLE STOP
OR GSB000  ; FOR EQUIPMENT DESIGN_ORDINARY TIMES ON
ANDLD
OUT W58.01  ; IND.SLIDE TRANSFER RET.
; rung 3
ILC(003)

### Section END
; rung 0
END(001)

## Program P16_ROTARY_TRANSFER (cyclic task 6)
Local symbols
GP1_ADV_RTN E0_47.03 BOOL
GP2_ADV_RTN E0_47.04 BOOL
Hold_GP1_ADV E0_47.01 BOOL
Hold_GP1_RET E0_47.02 BOOL
LB1399 E0_30.11 BOOL  ; P12 AutoCycleEnd
LB2000 E0_30.12 BOOL  ; AUTO START BEGIN
LB2001 E0_30.13 BOOL  ; GP2 STAND BY
LB2002 E0_30.14 BOOL  ; GP2 LOAD FINISH WORK
LB2003 E0_30.15 BOOL  ; GP2 UNLOAD UNFINISH WORK
LB2004 E0_31.00 BOOL  ; GP2 PROGRAM CONFIRM
LB2005 E0_31.01 BOOL  ; 1EC1 FORWARD START
LB2006 E0_31.02 BOOL  ; 1EC1 FORWARD COMPLETE
LB2007 E0_31.03 BOOL  ; SOL.GIPPER TRANSFER 1 CHUCK
LB2008 E0_31.04 BOOL  ; SOL.GIPPER TRANSFER 1 CHUCK CONF
LB2011 E0_31.05 BOOL  ; SOL.GIPPER TRANSFER 2 UNCHUCK
LB2012 E0_31.06 BOOL  ; SOL.GIPPER TRANSFER 2 UNCHUCK CONF
LB2013 E0_31.07 BOOL  ; GP2 UNLOAD CONF
LB2014 E0_31.08 BOOL  ; 1EC1 BACKWARD START
LB2015 E0_31.09 BOOL  ; 1EC1 BACKWARD START CONF
LB2016 E0_31.10 BOOL  ; AUTO START BEGIN
LB2017 E0_31.11 BOOL  ; FINAL CAULKING FULL WORK
LB2018 E0_31.12 BOOL  ; FINAL CAULKING NOT FULL
LB2019 E0_31.13 BOOL  ; 1EC1 FORWARD START
LB2020 E0_31.14 BOOL  ; 1EC1 FORWARD START CONF
LB2021 E0_31.15 BOOL  ; SOL.GIPPER TRANSFER 2 CHUCK
LB2022 E0_32.00 BOOL  ; SOL.GIPPER TRANSFER 2 CHUCK CONF
LB2023 E0_32.01 BOOL  ; 1EC1 BACKWARD START
LB2024 E0_32.02 BOOL  ; 1EC1 BACKWARD CONF
LB2025 E0_32.03 BOOL  ; 1EC2 FORWARD START
LB2026 E0_32.04 BOOL  ; 1EC2 FORWARD CONF
LB2027 E0_32.05 BOOL  ; SOL.GIPPER TRANSFER UNIT 2 ADV
LB2028 E0_32.06 BOOL  ; SOL.GIPPER TRANSFER UNIT 2 ADV CONF
LB2029 E0_32.07 BOOL  ; 1EC1 FORWARD START
LB2030 E0_32.08 BOOL  ; 1EC1 FORWARD START CONF
LB2031 E0_32.09 BOOL  ; SOL.GIPPER TRANSFER 1 UNCHUCK
LB2032 E0_32.10 BOOL  ; SOL.GIPPER TRANSFER 1 UNCHUCK CONF
LB2033 E0_32.11 BOOL  ; SOL.GIPPER TRANSFER 2 UNCHUCK
LB2034 E0_32.12 BOOL  ; SOL.GIPPER TRANSFER 2 UNCHUCK CONF
LB2035 E0_32.13 BOOL  ; 1EC1 BACKKWARD START
LB2036 E0_32.14 BOOL  ; 1EC1 BACKKWARD START CONF
LB2037 E0_32.15 BOOL  ; SOL.GIPPER TRANSFER UNIT 2 RET
LB2038 E0_33.00 BOOL  ; SOL.GIPPER TRANSFER UNIT 2 RET CONF
LB2042 E0_33.01 BOOL  ; 1EC2 FORWARD START
LB2043 E0_33.02 BOOL  ; 1EC2 FORWARD START CONF
LB2044 E0_33.03 BOOL  ; 1EC1 FORWARD START
LB2045 E0_33.04 BOOL  ; 1EC1 FORWARD START CONF
LB2046 E0_33.05 BOOL  ; SOL.GIPPER TRANSFER 1 UNCHUCK
LB2047 E0_33.06 BOOL  ; SOL.GIPPER TRANSFER 1 UNCHUCK CONF
LB2052 E0_33.07 BOOL  ; 1EC1 BACKWARD START
LB2053 E0_33.08 BOOL  ; 1EC1 BACKWARD START CONF
LB2054 E0_33.09 BOOL  ; 1EC2 BACKWARD START
LB2055 E0_33.10 BOOL  ; 1EC2 BACKWARD START CONF
LB2056 E0_33.11 BOOL  ; CYCLE STOP LOOP
LB2057 E0_33.12 BOOL  ; END MOTION
LB2058 E0_33.13 BOOL  ; 1EC2 BACKWARD START
LB2059 E0_33.14 BOOL  ; 1EC2 BACKWARD START CONF
LB2060 E0_33.15 BOOL  ; GRIPPER 1 LOAD FINISH
LB2061 E0_34.00 BOOL  ; GRIPPER 2 LOAD FINISH
LB2062 E0_34.01 BOOL  ; GP2 STAND BY
LB2063 E0_34.02 BOOL  ; GP2 LOAD UNFINISH
LB2064 E0_34.03 BOOL  ; AUTO BEGIN
LB2064A E0_49.15 BOOL  ; Cycle Stop
LB2065 E0_34.04 BOOL  ; 1EC1 FORWARD START
LB2066 E0_34.05 BOOL  ; 1EC1 FORWARD START CONF
LB2067 E0_34.06 BOOL  ; SOL.GIPPER TRANSFER 1 CHUCK
LB2068 E0_34.07 BOOL  ; SOL.GIPPER TRANSFER 2 CHUCK
LB2069 E0_34.08 BOOL  ; SOL.GIPPER TRANSFER 2 CHUCK CONF
LB2070 E0_34.09 BOOL  ; SOL.GIPPER TRANSFER 1 CHUCK CONF
LB2071 E0_34.10 BOOL  ; SOL.GIPPER TRANSFER 2 CHUCK
LB2072 E0_34.11 BOOL  ; SOL.GIPPER TRANSFER 2 CHUCK CONF
LB2073 E0_34.12 BOOL  ; GP1 STAND BY
LB2074 E0_34.13 BOOL  ; GP1 LOAD UNFINISH
LB2075 E0_34.14 BOOL  ; AUTO BEGIN
LB2075A E0_49.13 BOOL  ; Cycle Stop
LB2076 E0_34.15 BOOL  ; 1EC1 FORWARD START
LB2077 E0_35.00 BOOL  ; 1EC1 FORWARD START CONF
LB2078 E0_35.01 BOOL  ; SOL.GIPPER TRANSFER 2 CHUCK
LB2079 E0_35.02 BOOL  ; SOL.GIPPER TRANSFER 2 CHUCK CONF
LB2080 E0_35.03 BOOL  ; SOL.GIPPER TRANSFER 1 CHUCK
LB2081 E0_35.04 BOOL  ; SOL.GIPPER TRANSFER 1 CHUCK CONF
LB2082 E0_35.05 BOOL  ; GP1 END
LB2083 E0_35.06 BOOL  ; GP2 END
LB2084 E0_35.07 BOOL  ; 1EC1 BACKWARD START
LB2085 E0_35.08 BOOL  ; 1EC1 BACKWARD START CONF
LB2086 E0_35.09 BOOL  ; GRIPPER 1 UNLOAD
LB2087 E0_35.10 BOOL  ; GRIPPER 2 UNLOAD
LB2088 E0_35.11 BOOL  ; SOL.GIPPER TRANSFER UNIT 1 ADV
LB2089 E0_35.12 BOOL  ; SOL.GIPPER TRANSFER UNIT 1 ADV CONF
LB2090 E0_35.13 BOOL  ; 1EC1 FORWARD start (take in finish GP1)
LB2091 E0_35.14 BOOL  ; 1EC1 FORWARD START CONF
LB2092 E0_35.15 BOOL  ; SOL.GIPPER TRANSFER 1 UNCHUCK
LB2093 E0_36.00 BOOL  ; SOL.GIPPER TRANSFER 1 UNCHUCK CONF
LB2094 E0_36.01 BOOL  ; SOL.GIPPER TRANSFER 2 UNCHUCK
LB2095 E0_36.02 BOOL  ; SOL.GIPPER TRANSFER 2 UNCHUCK CONF
LB2097 E0_36.03 BOOL  ; SOL.GIPPER TRANSFER UNIT 2 ADV
LB2098 E0_36.04 BOOL  ; SOL.GIPPER TRANSFER UNIT 2 ADV CONF
LB2099 E0_36.05 BOOL  ; 1EC1 FORWARD start (take in finish GP2)
LB2100 E0_36.06 BOOL  ; 1EC1 FORWARD START CONF
LB2101 E0_36.07 BOOL  ; SOL.GIPPER TRANSFER 2 UNCHUCK
LB2102 E0_36.08 BOOL  ; SOL.GIPPER TRANSFER 2 UNCHUCK CONF
LB2103 E0_36.09 BOOL  ; SOL.GIPPER TRANSFER 1 UNCHUCK
LB2104 E0_36.10 BOOL  ; SOL.GIPPER TRANSFER 1 UNCHUCK CONF
LB2105 E0_36.11 BOOL  ; GP2 MAIN OP END
LB2106 E0_36.12 BOOL  ; 1EC1 BACKWARD START
LB2107 E0_36.13 BOOL  ; 1EC1 BACKWARD START CONF
LB2108 E0_36.14 BOOL  ; 1EC2 BACKWARD START
LB2109 E0_36.15 BOOL  ; 1EC2 BACKWARD START CONF
LB2110 E0_37.00 BOOL  ; 1EC2 FORWARD START
LB2110_1 E0_46.11 BOOL  ; EC2 backward
LB2111 E0_37.01 BOOL  ; 1EC2 FORWARD START CONF
LB2111_1 E0_47.11 BOOL  ; EC 2 backward confirm
LB2112 E0_37.02 BOOL  ; GRIPPER 1 UNLOAD
LB2113 E0_37.03 BOOL  ; GRIPPER 2 UNLOAD
LB2114 E0_37.04 BOOL  ; 1EC2 BACKWARD START
LB2115 E0_37.05 BOOL  ; 1EC2 BACKWARD START CONF
LB2116 E0_37.06 BOOL  ; SOL.GIPPER TRANSFER UNIT 1 ADV
LB2117 E0_37.07 BOOL  ; SOL.GIPPER TRANSFER UNIT 1 ADV CONF
LB2118 E0_37.08 BOOL  ; 1EC1 FORWARD START
LB2119 E0_37.09 BOOL  ; 1EC1 FORWARD START CONF
LB2120 E0_37.10 BOOL  ; SOL.GIPPER TRANSFER 1 UNCHUCK
LB2121 E0_37.11 BOOL  ; SOL.GIPPER TRANSFER 1 UNCHUCK CONF
LB2122 E0_37.12 BOOL  ; SOL.GIPPER TRANSFER 2 CHUCK
LB2123 E0_37.13 BOOL  ; SOL.GIPPER TRANSFER 2 CHUCK CONF
LB2124 E0_37.14 BOOL  ; GP1 MAIN OP END
LB2125 E0_37.15 BOOL  ; 1EC2 FORWARD START
LB2126 E0_38.00 BOOL  ; 1EC2 FORWARD START CONF
LB2127 E0_38.01 BOOL  ; SOL.GIPPER TRANSFER UNIT 2 ADV
LB2128 E0_38.02 BOOL  ; SOL.GIPPER TRANSFER UNIT 2 ADV CONF
LB2129 E0_38.03 BOOL  ; 1EC1 FORWARD START
LB2130 E0_38.04 BOOL  ; 1EC1 FORWARD START CONF
LB2131 E0_38.05 BOOL  ; SOL.GIPPER TRANSFER 2 UNCHUCK
LB2132 E0_38.06 BOOL  ; SOL.GIPPER TRANSFER 2 UNCHUCK CONF
LB2133 E0_38.07 BOOL  ; SOL.GIPPER TRANSFER 1 CHUCK
LB2134 E0_38.08 BOOL  ; SOL.GIPPER TRANSFER 1 CHUCK CONF
LB2135 E0_38.09 BOOL  ; GP2 MAIN OP END
LB2136 E0_38.10 BOOL  ; 1EC1 BACKWARD START
LB2137 E0_38.11 BOOL  ; 1EC1 BACKWARD START CONF
LB2140 E0_38.12 BOOL  ; SOL.GIPPER TRANSFER UNIT 1 RET
LB2141 E0_38.13 BOOL  ; SOL.GIPPER TRANSFER UNIT 1 RET CONF
LB2142 E0_38.14 BOOL  ; 1EC1 BACKWARD START
LB2143 E0_38.15 BOOL  ; 1EC1 BACKWARD START CONF
LB2144 E0_39.00 BOOL  ; SOL.GIPPER TRANSFER UNIT 2 RET
LB2145 E0_39.01 BOOL  ; SOL.GIPPER TRANSFER UNIT 2 RET
LB2150 E0_39.02 BOOL  ; 1EC1 BACKWARD START
LB2151 E0_39.03 BOOL  ; 1EC1 BACKWARD START CONF
LB2152 E0_39.04 BOOL  ; SOL.GIPPER TRANSFER UNIT 1 RET
LB2153 E0_39.05 BOOL  ; SOL.GIPPER TRANSFER UNIT 1 RET CONF
LB2154 E0_39.06 BOOL  ; SOL.GIPPER TRANSFER UNIT 2 RET
LB2155 E0_39.07 BOOL  ; SOL.GIPPER TRANSFER UNIT 2 RET CONF
LB2160 E0_39.08 BOOL  ; GP2 LOAD WORK
LB2161 E0_39.09 BOOL  ; GP2 STAND BY
LB2162 E0_39.10 BOOL  ; GP1 LOAD WORK
LB2163 E0_39.11 BOOL  ; GP1 STAND BY
LB2190 E0_39.12 BOOL  ; GP1 MAIN OP END
LB2194 E0_39.13 BOOL  ; P16 Cycle end Case5
LB2195 E0_39.14 BOOL  ; P16 Cycle end Case1
LB2196 E0_39.15 BOOL  ; P16 Cycle end Case2
LB2197 E0_40.00 BOOL  ; P16 Case3 End
LB2198 E0_40.01 BOOL  ; P16 Cycle end Case4
LB2199 E0_40.02 BOOL  ; P16 AutoCycleEnd
LB2341 E0_47.07 BOOL  ; start trigger condition
LB340 E0_40.03 BOOL  ; IND 1 CYCLE
LB566 E0_40.04 BOOL  ; Master OK operation
LB567 E0_40.05 BOOL  ; Master OK Complete
LB568 E0_40.06 BOOL  ; Master NG Operation
LB569 E0_40.07 BOOL  ; Master NG Complete
LB600 E0_40.08 BOOL  ; P16 CycleStart
LB601 E0_40.09 BOOL  ; Take out Raw work
LB602 E0_40.10 BOOL  ; Take In Raw Work
LB603 E0_40.11 BOOL  ; Take Out Finish Work
LB604 E0_40.12 BOOL  ; Take In Finish Work
LB605 E0_40.13 BOOL  ; P16 GP1 UNLoadFinish DISCHARGE WK
LB6325 E0_47.06 BOOL  ; unit started
LB6392 E0_40.14 BOOL  ; master check condition
LB6393 E0_40.15 BOOL  ; normal operation
LT123 T3025 TIMER  ; safety timer
LT324 T3026 TIMER
dbug2 E0_41.00 BOOL
dbug3 E0_41.01 BOOL
e0_3200_00 E0_46.12 BOOL

### Section HMI_Output

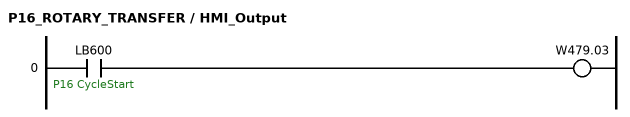
; rung 0
LD LB600  ; P16 CycleStart
OUT W479.03

### Section Autorun

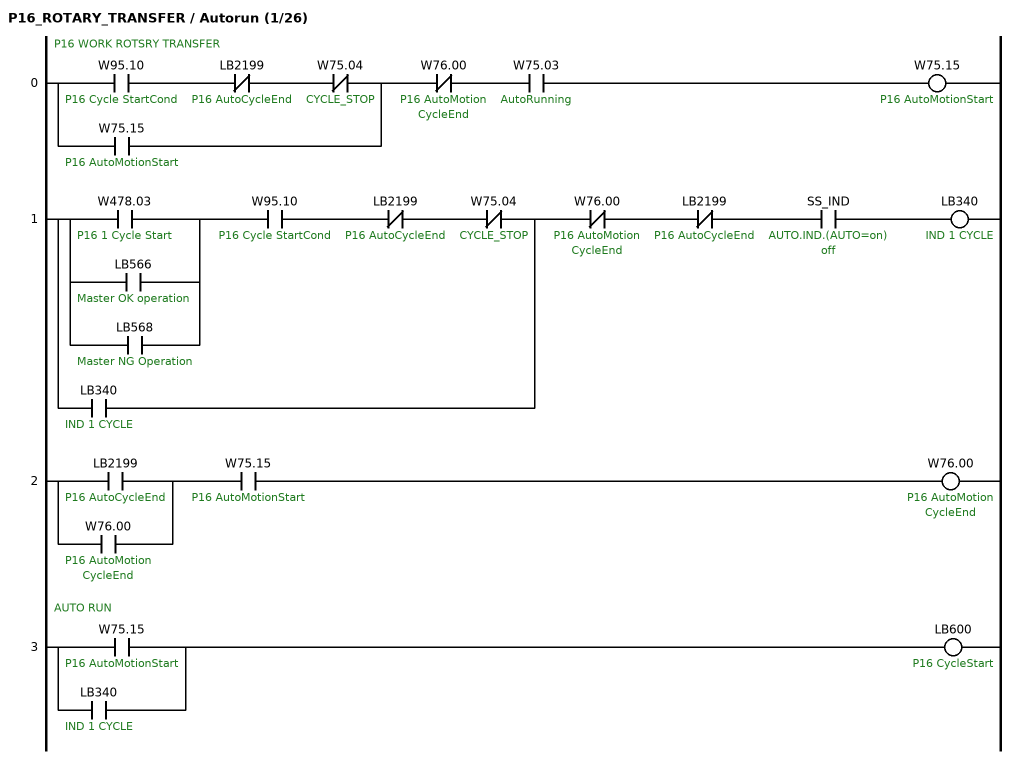
; rung 0: P16 WORK ROTSRY TRANSFER
LD W95.10  ; P16 Cycle StartCond
ANDNOT LB2199  ; P16 AutoCycleEnd
ANDNOT W75.04  ; CYCLE_STOP
OR W75.15  ; P16 AutoMotionStart
ANDNOT W76.00  ; P16 AutoMotion CycleEnd
AND W75.03  ; AutoRunning
OUT W75.15  ; P16 AutoMotionStart
; rung 1
LD W478.03  ; P16 1 Cycle Start
OR LB566  ; Master OK operation
OR LB568  ; Master NG Operation
AND W95.10  ; P16 Cycle StartCond
ANDNOT LB2199  ; P16 AutoCycleEnd
ANDNOT W75.04  ; CYCLE_STOP
OR LB340  ; IND 1 CYCLE
ANDNOT W76.00  ; P16 AutoMotion CycleEnd
ANDNOT LB2199  ; P16 AutoCycleEnd
AND SS_IND  ; AUTO.IND.(AUTO=on) off
OUT LB340  ; IND 1 CYCLE
; rung 2
LD LB2199  ; P16 AutoCycleEnd
OR W76.00  ; P16 AutoMotion CycleEnd
AND W75.15  ; P16 AutoMotionStart
OUT W76.00  ; P16 AutoMotion CycleEnd
; rung 3: AUTO RUN
LD W75.15  ; P16 AutoMotionStart
OR LB340  ; IND 1 CYCLE
OUT LB600  ; P16 CycleStart

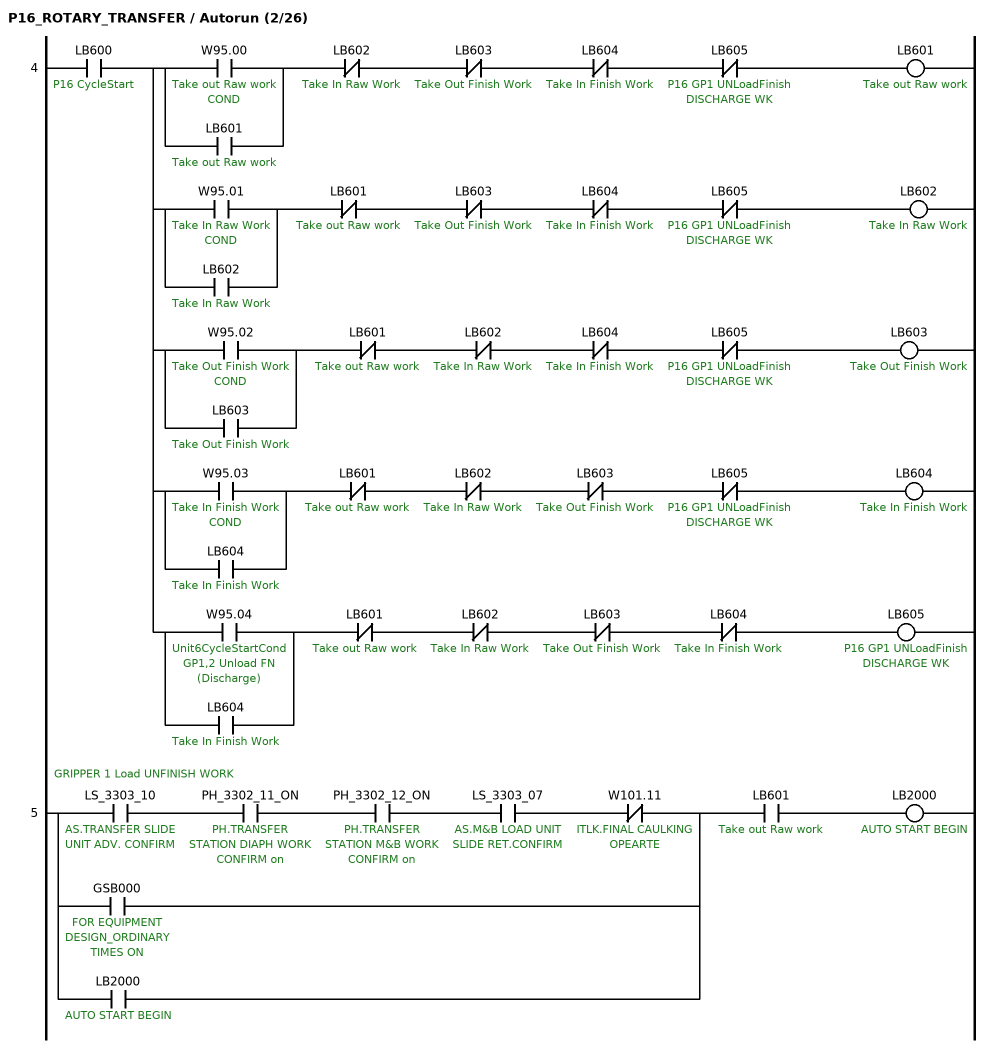
; rung 4
LD LB600  ; P16 CycleStart
OUT TR0
LD W95.00  ; Take out Raw work COND
OR LB601  ; Take out Raw work
ANDLD
ANDNOT LB602  ; Take In Raw Work
ANDNOT LB603  ; Take Out Finish Work
ANDNOT LB604  ; Take In Finish Work
ANDNOT LB605  ; P16 GP1 UNLoadFinish DISCHARGE WK
OUT LB601  ; Take out Raw work
LD TR0
LD W95.01  ; Take In Raw Work COND
OR LB602  ; Take In Raw Work
ANDLD
ANDNOT LB601  ; Take out Raw work
ANDNOT LB603  ; Take Out Finish Work
ANDNOT LB604  ; Take In Finish Work
ANDNOT LB605  ; P16 GP1 UNLoadFinish DISCHARGE WK
OUT LB602  ; Take In Raw Work
LD TR0
LD W95.02  ; Take Out Finish Work COND
OR LB603  ; Take Out Finish Work
ANDLD
ANDNOT LB601  ; Take out Raw work
ANDNOT LB602  ; Take In Raw Work
ANDNOT LB604  ; Take In Finish Work
ANDNOT LB605  ; P16 GP1 UNLoadFinish DISCHARGE WK
OUT LB603  ; Take Out Finish Work
LD TR0
LD W95.03  ; Take In Finish Work COND
OR LB604  ; Take In Finish Work
ANDLD
ANDNOT LB601  ; Take out Raw work
ANDNOT LB602  ; Take In Raw Work
ANDNOT LB603  ; Take Out Finish Work
ANDNOT LB605  ; P16 GP1 UNLoadFinish DISCHARGE WK
OUT LB604  ; Take In Finish Work
LD TR0
LD W95.04  ; Unit6CycleStartCond GP1,2 Unload FN (Discharge)
OR LB604  ; Take In Finish Work
ANDLD
ANDNOT LB601  ; Take out Raw work
ANDNOT LB602  ; Take In Raw Work
ANDNOT LB603  ; Take Out Finish Work
ANDNOT LB604  ; Take In Finish Work
OUT LB605  ; P16 GP1 UNLoadFinish DISCHARGE WK
; rung 5: GRIPPER 1 Load UNFINISH WORK
LD LS_3303_10  ; AS.TRANSFER SLIDE UNIT ADV. CONFIRM
AND PH_3302_11_ON  ; PH.TRANSFER STATION DIAPH WORK CONFIRM on
AND PH_3302_12_ON  ; PH.TRANSFER STATION M&B WORK CONFIRM on
AND LS_3303_07  ; AS.M&B LOAD UNIT SLIDE RET.CONFIRM
ANDNOT W101.11  ; ITLK.FINAL CAULKING OPEARTE
OR GSB000  ; FOR EQUIPMENT DESIGN_ORDINARY TIMES ON
OR LB2000  ; AUTO START BEGIN
AND LB601  ; Take out Raw work
OUT LB2000  ; AUTO START BEGIN

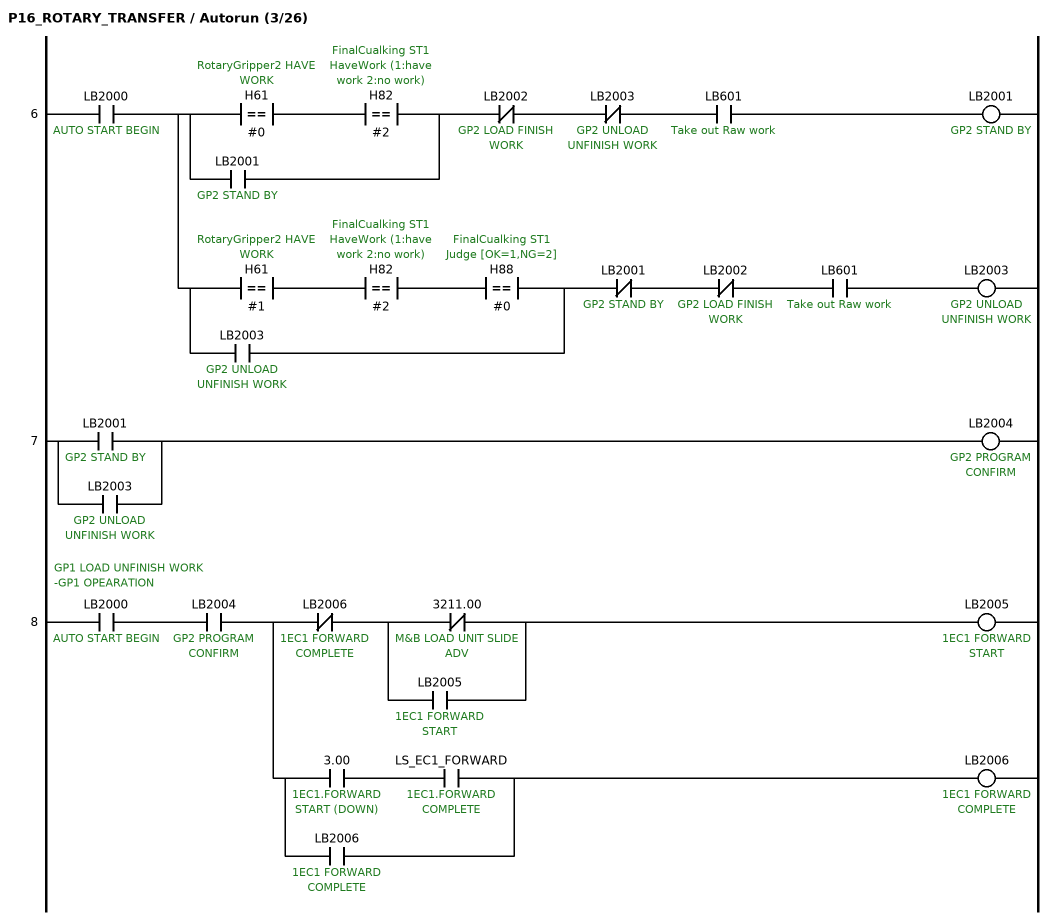
; rung 6
LD LB2000  ; AUTO START BEGIN
OUT TR0
LD=(300) H61 #0  ; RotaryGripper2 HAVE WORK
AND=(300) H82 #2  ; FinalCualking ST1 HaveWork (1:have work 2:no work)
OR LB2001  ; GP2 STAND BY
ANDLD
ANDNOT LB2002  ; GP2 LOAD FINISH WORK
ANDNOT LB2003  ; GP2 UNLOAD UNFINISH WORK
AND LB601  ; Take out Raw work
OUT LB2001  ; GP2 STAND BY
LD TR0
LD=(300) H61 #1  ; RotaryGripper2 HAVE WORK
AND=(300) H82 #2  ; FinalCualking ST1 HaveWork (1:have work 2:no work)
AND=(300) H88 #0  ; FinalCualking ST1 Judge [OK=1,NG=2]
OR LB2003  ; GP2 UNLOAD UNFINISH WORK
ANDLD
ANDNOT LB2001  ; GP2 STAND BY
ANDNOT LB2002  ; GP2 LOAD FINISH WORK
AND LB601  ; Take out Raw work
OUT LB2003  ; GP2 UNLOAD UNFINISH WORK
; rung 7
LD LB2001  ; GP2 STAND BY
OR LB2003  ; GP2 UNLOAD UNFINISH WORK
OUT LB2004  ; GP2 PROGRAM CONFIRM
; rung 8: GP1 LOAD UNFINISH WORK / -GP1 OPEARATION
LD LB2000  ; AUTO START BEGIN
AND LB2004  ; GP2 PROGRAM CONFIRM
OUT TR0
ANDNOT LB2006  ; 1EC1 FORWARD COMPLETE
LDNOT 3211.00  ; M&B LOAD UNIT SLIDE ADV
OR LB2005  ; 1EC1 FORWARD START
ANDLD
OUT LB2005  ; 1EC1 FORWARD START
LD TR0
LD 3.00  ; 1EC1.FORWARD START (DOWN)
AND LS_EC1_FORWARD  ; 1EC1.FORWARD COMPLETE
OR LB2006  ; 1EC1 FORWARD COMPLETE
ANDLD
OUT LB2006  ; 1EC1 FORWARD COMPLETE

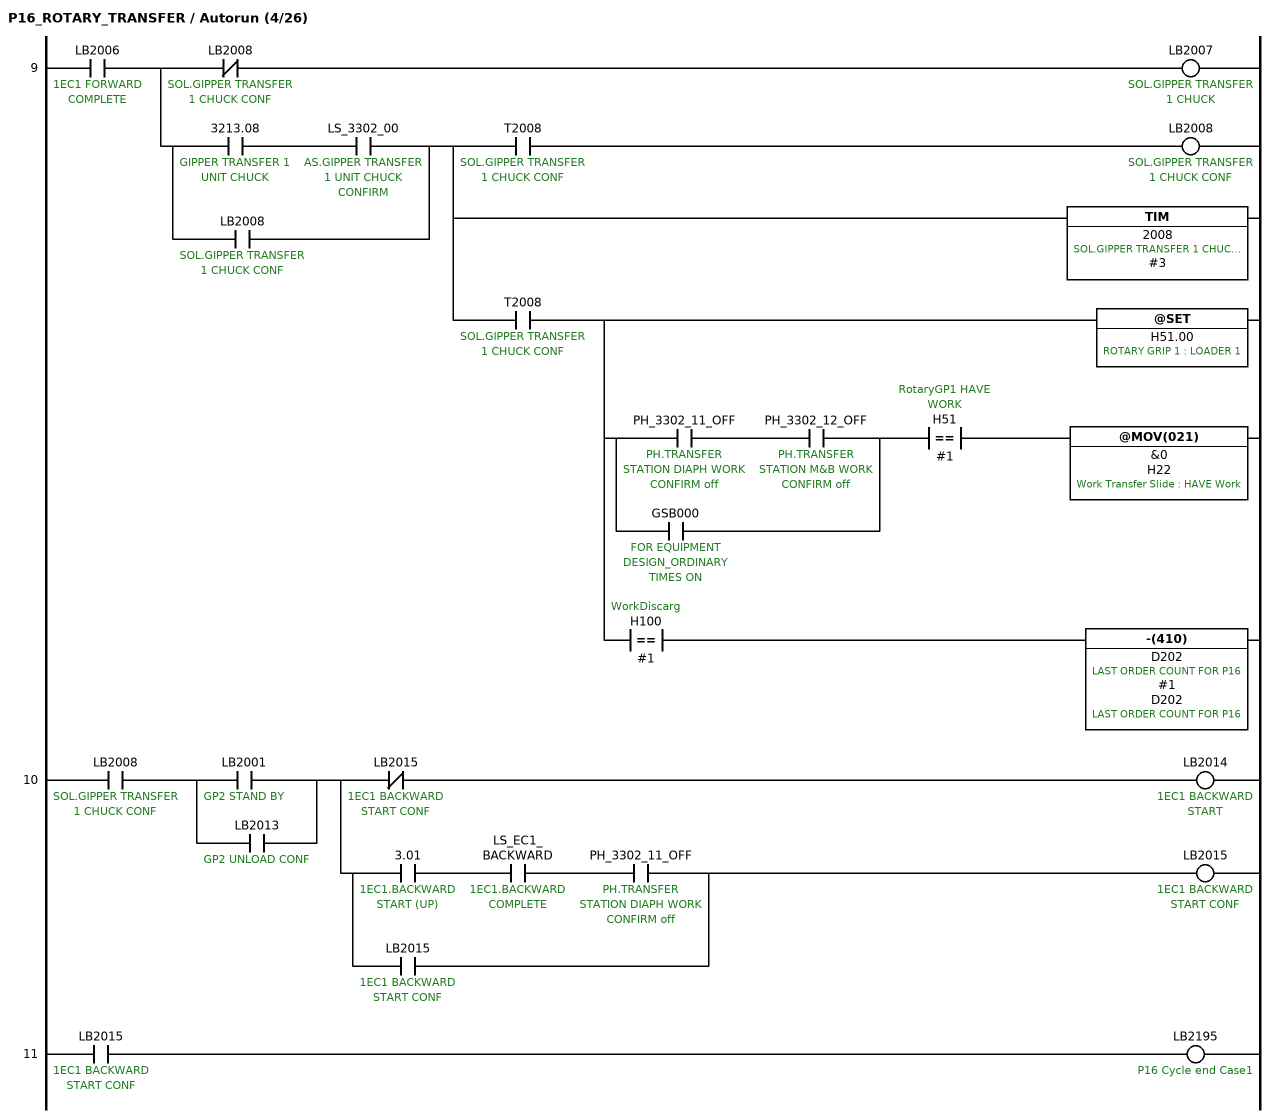
; rung 9
LD LB2006  ; 1EC1 FORWARD COMPLETE
OUT TR0
ANDNOT LB2008  ; SOL.GIPPER TRANSFER 1 CHUCK CONF
OUT LB2007  ; SOL.GIPPER TRANSFER 1 CHUCK
LD TR0
LD 3213.08  ; GIPPER TRANSFER 1 UNIT CHUCK
AND LS_3302_00  ; AS.GIPPER TRANSFER 1 UNIT CHUCK CONFIRM
OR LB2008  ; SOL.GIPPER TRANSFER 1 CHUCK CONF
ANDLD
OUT TR0
AND T2008  ; SOL.GIPPER TRANSFER 1 CHUCK CONF
OUT LB2008  ; SOL.GIPPER TRANSFER 1 CHUCK CONF
LD TR0
TIM 2008 #3  ; SOL.GIPPER TRANSFER 1 CHUCK CONF
AND T2008  ; SOL.GIPPER TRANSFER 1 CHUCK CONF
OUT TR0
@SET H51.00  ; ROTARY GRIP 1 : LOADER 1
LD PH_3302_11_OFF  ; PH.TRANSFER STATION DIAPH WORK CONFIRM off
AND PH_3302_12_OFF  ; PH.TRANSFER STATION M&B WORK CONFIRM off
OR GSB000  ; FOR EQUIPMENT DESIGN_ORDINARY TIMES ON
ANDLD
AND=(300) H51 #1  ; RotaryGP1 HAVE WORK
@MOV(021) &0 H22  ; Work Transfer Slide : HAVE Work
LD TR0
AND=(300) H100 #1  ; WorkDiscarg
-(410) D202 #1 D202  ; LAST ORDER COUNT FOR P16
; rung 10
LD LB2008  ; SOL.GIPPER TRANSFER 1 CHUCK CONF
LD LB2001  ; GP2 STAND BY
OR LB2013  ; GP2 UNLOAD CONF
ANDLD
OUT TR0
ANDNOT LB2015  ; 1EC1 BACKWARD START CONF
OUT LB2014  ; 1EC1 BACKWARD START
LD TR0
LD 3.01  ; 1EC1.BACKWARD START (UP)
AND LS_EC1_BACKWARD  ; 1EC1.BACKWARD COMPLETE
AND PH_3302_11_OFF  ; PH.TRANSFER STATION DIAPH WORK CONFIRM off
OR LB2015  ; 1EC1 BACKWARD START CONF
ANDLD
OUT LB2015  ; 1EC1 BACKWARD START CONF
; rung 11
LD LB2015  ; 1EC1 BACKWARD START CONF
OUT LB2195  ; P16 Cycle end Case1

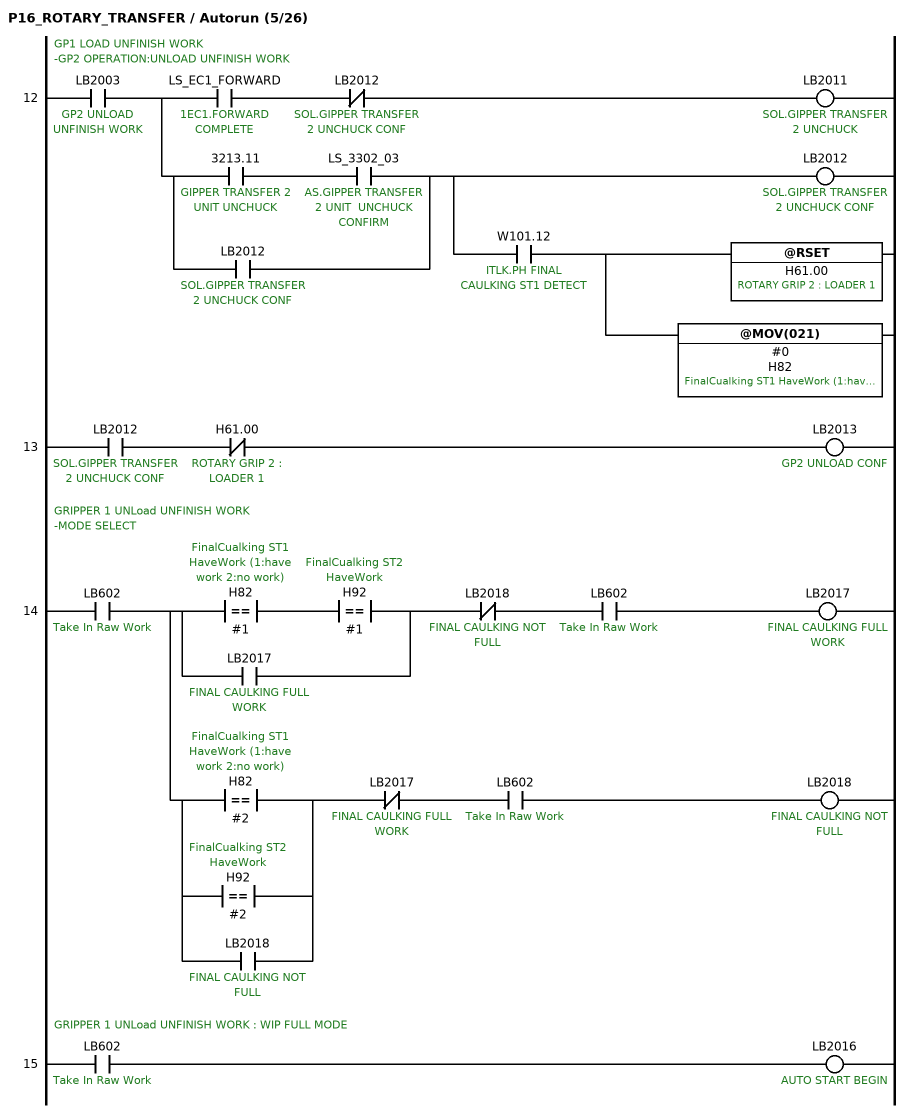
; rung 12: GP1 LOAD UNFINISH WORK / -GP2 OPERATION:UNLOAD UNFINISH WORK
LD LB2003  ; GP2 UNLOAD UNFINISH WORK
OUT TR0
AND LS_EC1_FORWARD  ; 1EC1.FORWARD COMPLETE
ANDNOT LB2012  ; SOL.GIPPER TRANSFER 2 UNCHUCK CONF
OUT LB2011  ; SOL.GIPPER TRANSFER 2 UNCHUCK
LD TR0
LD 3213.11  ; GIPPER TRANSFER 2 UNIT UNCHUCK
AND LS_3302_03  ; AS.GIPPER TRANSFER 2 UNIT  UNCHUCK CONFIRM
OR LB2012  ; SOL.GIPPER TRANSFER 2 UNCHUCK CONF
ANDLD
OUT LB2012  ; SOL.GIPPER TRANSFER 2 UNCHUCK CONF
AND W101.12  ; ITLK.PH FINAL CAULKING ST1 DETECT
@RSET H61.00  ; ROTARY GRIP 2 : LOADER 1
@MOV(021) #0 H82  ; FinalCualking ST1 HaveWork (1:have work 2:no work)
; rung 13
LD LB2012  ; SOL.GIPPER TRANSFER 2 UNCHUCK CONF
ANDNOT H61.00  ; ROTARY GRIP 2 : LOADER 1
OUT LB2013  ; GP2 UNLOAD CONF
; rung 14: GRIPPER 1 UNLoad UNFINISH WORK / -MODE SELECT
LD LB602  ; Take In Raw Work
OUT TR0
LD=(300) H82 #1  ; FinalCualking ST1 HaveWork (1:have work 2:no work)
AND=(300) H92 #1  ; FinalCualking ST2 HaveWork
OR LB2017  ; FINAL CAULKING FULL WORK
ANDLD
ANDNOT LB2018  ; FINAL CAULKING NOT FULL
AND LB602  ; Take In Raw Work
OUT LB2017  ; FINAL CAULKING FULL WORK
LD TR0
LD=(300) H82 #2  ; FinalCualking ST1 HaveWork (1:have work 2:no work)
OR=(300) H92 #2  ; FinalCualking ST2 HaveWork
OR LB2018  ; FINAL CAULKING NOT FULL
ANDLD
ANDNOT LB2017  ; FINAL CAULKING FULL WORK
AND LB602  ; Take In Raw Work
OUT LB2018  ; FINAL CAULKING NOT FULL
; rung 15: GRIPPER 1 UNLoad UNFINISH WORK : WIP FULL MODE
LD LB602  ; Take In Raw Work
OUT LB2016  ; AUTO START BEGIN

